   1:  PR[GP1:91,2] = PR[GP1:90,2] + 0.287;
   1:L PR[91] 10mm/sec CNT100;
   1:  PR[GP1:91,1] = PR[GP1:90,1] + -53.304;
   1:  PR[GP1:91,2] = PR[GP1:90,2] + -9.649;
   1:L PR[91] 10mm/sec CNT100;
   1:  PR[GP1:91,1] = PR[GP1:90,1] + -52.837;
   1:  PR[GP1:91,2] = PR[GP1:90,2] + -13.000;
   1:L PR[91] 10mm/sec CNT100;
   1:  PR[GP1:91,1] = PR[GP1:90,1] + -51.484;
   1:  PR[GP1:91,2] = PR[GP1:90,2] + -16.066;
   1:L PR[91] 10mm/sec CNT100;
   1:  PR[GP1:91,1] = PR[GP1:90,1] + -46.658;
   1:  PR[GP1:91,2] = PR[GP1:90,2] + -24.961;
   1:L PR[91] 10mm/sec CNT100;
   1:  PR[GP1:91,1] = PR[GP1:90,1] + -44.364;
   1:  PR[GP1:91,2] = PR[GP1:90,2] + -27.724;
   1:L PR[91] 10mm/sec CNT100;
   1:  PR[GP1:91,1] = PR[GP1:90,1] + -37.102;
   1:  PR[GP1:91,2] = PR[GP1:90,2] + -34.467;
   1:L PR[91] 10mm/sec CNT100;
   1:  PR[GP1:91,1] = PR[GP1:90,1] + -32.633;
   1:  PR[GP1:91,2] = PR[GP1:90,2] + -37.235;
   1:L PR[91] 10mm/sec CNT100;
   1:  PR[GP1:91,1] = PR[GP1:90,1] + -23.806;
   1:  PR[GP1:91,2] = PR[GP1:90,2] + -41.267;
   1:L PR[91] 10mm/sec CNT100;
   1:  PR[GP1:91,1] = PR[GP1:90,1] + -18.131;
   1:  PR[GP1:91,2] = PR[GP1:90,2] + -42.329;
   1:L PR[91] 10mm/sec CNT100;
   1:  PR[GP1:91,1] = PR[GP1:90,1] + -8.768;
   1:  PR[GP1:91,2] = PR[GP1:90,2] + -43.356;
   1:L PR[91] 10mm/sec CNT100;
   1:  PR[GP1:91,1] = PR[GP1:90,1] + -2.914;
   1:  PR[GP1:91,2] = PR[GP1:90,2] + -42.375;
   1:L PR[91] 10mm/sec CNT100;
   1:  PR[GP1:91,1] = PR[GP1:90,1] + -0.261;
   1:  PR[GP1:91,2] = PR[GP1:90,2] + -41.804;
   1:L PR[91] 10mm/sec CNT100;
   1:  PR[GP1:91,1] = PR[GP1:90,1] + 1.954;
   1:  PR[GP1:91,2] = PR[GP1:90,2] + -42.461;
   1:  PR[GP1:91,3] = PR[GP1:90,3] + 101.565;
   1:L PR[91] 10mm/sec CNT100;
   1:  PR[GP1:91,1] = PR[GP1:90,1] + 8.050;
   1:  PR[GP1:91,2] = PR[GP1:90,2] + -43.485;
   1:L PR[91] 10mm/sec CNT100;
   1:  PR[GP1:91,1] = PR[GP1:90,1] + 17.201;
   1:  PR[GP1:91,2] = PR[GP1:90,2] + -42.479;
   1:L PR[91] 10mm/sec CNT100;
   1:  PR[GP1:91,1] = PR[GP1:90,1] + 23.153;
   1:  PR[GP1:91,2] = PR[GP1:90,2] + -41.367;
   1:L PR[91] 10mm/sec CNT100;
   1:  PR[GP1:91,1] = PR[GP1:90,1] + 31.780;
   1:  PR[GP1:91,2] = PR[GP1:90,2] + -37.429;
   1:L PR[91] 10mm/sec CNT100;
   1:  PR[GP1:91,1] = PR[GP1:90,1] + 36.498;
   1:  PR[GP1:91,2] = PR[GP1:90,2] + -34.507;
   1:L PR[91] 10mm/sec CNT100;
   1:  PR[GP1:91,1] = PR[GP1:90,1] + 43.596;
   1:  PR[GP1:91,2] = PR[GP1:90,2] + -27.908;
   1:L PR[91] 10mm/sec CNT100;
   1:  PR[GP1:91,1] = PR[GP1:90,1] + 46.034;
   1:  PR[GP1:91,2] = PR[GP1:90,2] + -24.972;
   1:L PR[91] 10mm/sec CNT100;
   1:  PR[GP1:91,1] = PR[GP1:90,1] + 50.751;
   1:  PR[GP1:91,2] = PR[GP1:90,2] + -16.292;
   1:L PR[91] 10mm/sec CNT100;
   1:  PR[GP1:91,1] = PR[GP1:90,1] + 52.201;
   1:  PR[GP1:91,2] = PR[GP1:90,2] + -13.008;
   1:L PR[91] 10mm/sec CNT100;
   1:  PR[GP1:91,1] = PR[GP1:90,1] + 53.844;
   1:  PR[GP1:91,2] = PR[GP1:90,2] + -3.236;
   1:L PR[91] 10mm/sec CNT100;
   1:  PR[GP1:91,1] = PR[GP1:90,1] + 53.846;
   1:  PR[GP1:91,2] = PR[GP1:90,2] + -2.997;
   1:L PR[91] 10mm/sec CNT100;
   1:  PR[GP1:91,1] = PR[GP1:90,1] + 54.302;
   1:  PR[GP1:91,2] = PR[GP1:90,2] + 0.271;
   1:L PR[91] 10mm/sec CNT100;
   1:  PR[GP1:91,1] = PR[GP1:90,1] + 52.690;
   1:  PR[GP1:91,2] = PR[GP1:90,2] + 10.014;
   1:L PR[91] 10mm/sec CNT100;
   1:  PR[GP1:91,1] = PR[GP1:90,1] + 52.191;
   1:  PR[GP1:91,2] = PR[GP1:90,2] + 13.594;
   1:L PR[91] 10mm/sec CNT100;
   1:  PR[GP1:91,1] = PR[GP1:90,1] + 50.744;
   1:  PR[GP1:91,2] = PR[GP1:90,2] + 16.870;
   1:L PR[91] 10mm/sec CNT100;
   1:  PR[GP1:91,1] = PR[GP1:90,1] + 46.008;
   1:  PR[GP1:91,2] = PR[GP1:90,2] + 25.563;
   1:L PR[91] 10mm/sec CNT100;
   1:  PR[GP1:91,1] = PR[GP1:90,1] + 43.570;
   1:  PR[GP1:91,2] = PR[GP1:90,2] + 28.500;
   1:L PR[91] 10mm/sec CNT100;
   1:  PR[GP1:91,1] = PR[GP1:90,1] + 36.447;
   1:  PR[GP1:91,2] = PR[GP1:90,2] + 35.099;
   1:L PR[91] 10mm/sec CNT100;
   1:  PR[GP1:91,1] = PR[GP1:90,1] + 31.727;
   1:  PR[GP1:91,2] = PR[GP1:90,2] + 38.022;
   1:L PR[91] 10mm/sec CNT100;
   1:  PR[GP1:91,1] = PR[GP1:90,1] + 23.077;
   1:  PR[GP1:91,2] = PR[GP1:90,2] + 41.946;
   1:L PR[91] 10mm/sec CNT100;
   1:  PR[GP1:91,1] = PR[GP1:90,1] + 17.121;
   1:  PR[GP1:91,2] = PR[GP1:90,2] + 43.059;
   1:L PR[91] 10mm/sec CNT100;
   1:  PR[GP1:91,1] = PR[GP1:90,1] + 7.957;
   1:  PR[GP1:91,2] = PR[GP1:90,2] + 44.038;
   1:L PR[91] 10mm/sec CNT100;
   1:  PR[GP1:91,1] = PR[GP1:90,1] + -0.260;
   1:  PR[GP1:91,2] = PR[GP1:90,2] + 42.592;
   1:L PR[91] 10mm/sec CNT100;
   1:  PR[GP1:91,1] = PR[GP1:90,1] + -8.486;
   1:  PR[GP1:91,2] = PR[GP1:90,2] + 44.037;
   1:L PR[91] 10mm/sec CNT100;
   1:  PR[GP1:91,1] = PR[GP1:90,1] + -17.650;
   1:  PR[GP1:91,2] = PR[GP1:90,2] + 43.060;
   1:L PR[91] 10mm/sec CNT100;
   1:  PR[GP1:91,1] = PR[GP1:90,1] + -23.604;
   1:  PR[GP1:91,2] = PR[GP1:90,2] + 41.946;
   1:L PR[91] 10mm/sec CNT100;
   1:  PR[GP1:91,1] = PR[GP1:90,1] + -32.254;
   1:  PR[GP1:91,2] = PR[GP1:90,2] + 38.019;
   1:L PR[91] 10mm/sec CNT100;
   1:  PR[GP1:91,1] = PR[GP1:90,1] + -36.973;
   1:  PR[GP1:91,2] = PR[GP1:90,2] + 35.097;
   1:L PR[91] 10mm/sec CNT100;
   1:  PR[GP1:91,1] = PR[GP1:90,1] + -44.096;
   1:  PR[GP1:91,2] = PR[GP1:90,2] + 28.506;
   1:L PR[91] 10mm/sec CNT100;
   1:  PR[GP1:91,1] = PR[GP1:90,1] + -46.534;
   1:  PR[GP1:91,2] = PR[GP1:90,2] + 25.569;
   1:L PR[91] 10mm/sec CNT100;
   1:  PR[GP1:91,1] = PR[GP1:90,1] + -51.270;
   1:  PR[GP1:91,2] = PR[GP1:90,2] + 16.861;
   1:L PR[91] 10mm/sec CNT100;
   1:  PR[GP1:91,1] = PR[GP1:90,1] + -52.721;
   1:  PR[GP1:91,2] = PR[GP1:90,2] + 13.576;
   1:L PR[91] 10mm/sec CNT100;
   1:  PR[GP1:91,1] = PR[GP1:90,1] + -54.370;
   1:  PR[GP1:91,2] = PR[GP1:90,2] + 3.794;
   1:L PR[91] 10mm/sec CNT100;
   1:  PR[GP1:91,1] = PR[GP1:90,1] + -54.373;
   1:  PR[GP1:91,2] = PR[GP1:90,2] + 3.555;
   1:L PR[91] 10mm/sec CNT100;
   1:  PR[GP1:91,1] = PR[GP1:90,1] + -54.828;
   1:  PR[GP1:91,2] = PR[GP1:90,2] + 0.287;
   1:L PR[91] 10mm/sec CNT100;
   1:  PR[GP1:91,1] = PR[GP1:90,1] + -53.223;
   1:  PR[GP1:91,2] = PR[GP1:90,2] + -9.426;
   1:L PR[91] 10mm/sec CNT100;
   1:  PR[GP1:91,1] = PR[GP1:90,1] + -52.724;
   1:  PR[GP1:91,2] = PR[GP1:90,2] + -13.005;
   1:L PR[91] 10mm/sec CNT100;
   1:  PR[GP1:91,1] = PR[GP1:90,1] + -51.277;
   1:  PR[GP1:91,2] = PR[GP1:90,2] + -16.282;
   1:L PR[91] 10mm/sec CNT100;
   1:  PR[GP1:91,1] = PR[GP1:90,1] + -46.560;
   1:  PR[GP1:91,2] = PR[GP1:90,2] + -24.978;
   1:L PR[91] 10mm/sec CNT100;
   1:  PR[GP1:91,1] = PR[GP1:90,1] + -44.122;
   1:  PR[GP1:91,2] = PR[GP1:90,2] + -27.914;
   1:L PR[91] 10mm/sec CNT100;
   1:  PR[GP1:91,1] = PR[GP1:90,1] + -37.024;
   1:  PR[GP1:91,2] = PR[GP1:90,2] + -34.505;
   1:L PR[91] 10mm/sec CNT100;
   1:  PR[GP1:91,1] = PR[GP1:90,1] + -32.308;
   1:  PR[GP1:91,2] = PR[GP1:90,2] + -37.426;
   1:L PR[91] 10mm/sec CNT100;
   1:  PR[GP1:91,1] = PR[GP1:90,1] + -23.680;
   1:  PR[GP1:91,2] = PR[GP1:90,2] + -41.367;
   1:L PR[91] 10mm/sec CNT100;
   1:  PR[GP1:91,1] = PR[GP1:90,1] + -17.730;
   1:  PR[GP1:91,2] = PR[GP1:90,2] + -42.480;
   1:L PR[91] 10mm/sec CNT100;
   1:  PR[GP1:91,1] = PR[GP1:90,1] + -8.579;
   1:  PR[GP1:91,2] = PR[GP1:90,2] + -43.484;
   1:L PR[91] 10mm/sec CNT100;
   1:  PR[GP1:91,1] = PR[GP1:90,1] + -2.476;
   1:  PR[GP1:91,2] = PR[GP1:90,2] + -42.461;
   1:L PR[91] 10mm/sec CNT100;
   1:  PR[GP1:91,1] = PR[GP1:90,1] + -0.261;
   1:  PR[GP1:91,2] = PR[GP1:90,2] + -41.985;
   1:L PR[91] 10mm/sec CNT100;
   1:  PR[GP1:91,1] = PR[GP1:90,1] + 1.516;
   1:  PR[GP1:91,2] = PR[GP1:90,2] + -42.548;
   1:  PR[GP1:91,3] = PR[GP1:90,3] + 102.175;
   1:L PR[91] 10mm/sec CNT100;
   1:  PR[GP1:91,1] = PR[GP1:90,1] + 7.860;
   1:  PR[GP1:91,2] = PR[GP1:90,2] + -43.613;
   1:L PR[91] 10mm/sec CNT100;
   1:  PR[GP1:91,1] = PR[GP1:90,1] + 16.800;
   1:  PR[GP1:91,2] = PR[GP1:90,2] + -42.631;
   1:L PR[91] 10mm/sec CNT100;
   1:  PR[GP1:91,1] = PR[GP1:90,1] + 23.027;
   1:  PR[GP1:91,2] = PR[GP1:90,2] + -41.467;
   1:L PR[91] 10mm/sec CNT100;
   1:  PR[GP1:91,1] = PR[GP1:90,1] + 31.455;
   1:  PR[GP1:91,2] = PR[GP1:90,2] + -37.620;
   1:L PR[91] 10mm/sec CNT100;
   1:  PR[GP1:91,1] = PR[GP1:90,1] + 36.419;
   1:  PR[GP1:91,2] = PR[GP1:90,2] + -34.545;
   1:L PR[91] 10mm/sec CNT100;
   1:  PR[GP1:91,1] = PR[GP1:90,1] + 43.355;
   1:  PR[GP1:91,2] = PR[GP1:90,2] + -28.098;
   1:L PR[91] 10mm/sec CNT100;
   1:  PR[GP1:91,1] = PR[GP1:90,1] + 45.936;
   1:  PR[GP1:91,2] = PR[GP1:90,2] + -24.988;
   1:L PR[91] 10mm/sec CNT100;
   1:  PR[GP1:91,1] = PR[GP1:90,1] + 50.545;
   1:  PR[GP1:91,2] = PR[GP1:90,2] + -16.509;
   1:L PR[91] 10mm/sec CNT100;
   1:  PR[GP1:91,1] = PR[GP1:90,1] + 52.088;
   1:  PR[GP1:91,2] = PR[GP1:90,2] + -13.013;
   1:L PR[91] 10mm/sec CNT100;
   1:  PR[GP1:91,1] = PR[GP1:90,1] + 53.693;
   1:  PR[GP1:91,2] = PR[GP1:90,2] + -3.467;
   1:L PR[91] 10mm/sec CNT100;
   1:  PR[GP1:91,1] = PR[GP1:90,1] + 53.695;
   1:  PR[GP1:91,2] = PR[GP1:90,2] + -3.233;
   1:L PR[91] 10mm/sec CNT100;
   1:  PR[GP1:91,1] = PR[GP1:90,1] + 54.184;
   1:  PR[GP1:91,2] = PR[GP1:90,2] + 0.271;
   1:L PR[91] 10mm/sec CNT100;
   1:  PR[GP1:91,1] = PR[GP1:90,1] + 52.609;
   1:  PR[GP1:91,2] = PR[GP1:90,2] + 9.790;
   1:L PR[91] 10mm/sec CNT100;
   1:  PR[GP1:91,1] = PR[GP1:90,1] + 52.078;
   1:  PR[GP1:91,2] = PR[GP1:90,2] + 13.598;
   1:L PR[91] 10mm/sec CNT100;
   1:  PR[GP1:91,1] = PR[GP1:90,1] + 50.538;
   1:  PR[GP1:91,2] = PR[GP1:90,2] + 17.086;
   1:L PR[91] 10mm/sec CNT100;
   1:  PR[GP1:91,1] = PR[GP1:90,1] + 45.911;
   1:  PR[GP1:91,2] = PR[GP1:90,2] + 25.579;
   1:L PR[91] 10mm/sec CNT100;
   1:  PR[GP1:91,1] = PR[GP1:90,1] + 43.329;
   1:  PR[GP1:91,2] = PR[GP1:90,2] + 28.690;
   1:L PR[91] 10mm/sec CNT100;
   1:  PR[GP1:91,1] = PR[GP1:90,1] + 36.370;
   1:  PR[GP1:91,2] = PR[GP1:90,2] + 35.136;
   1:L PR[91] 10mm/sec CNT100;
   1:  PR[GP1:91,1] = PR[GP1:90,1] + 31.403;
   1:  PR[GP1:91,2] = PR[GP1:90,2] + 38.212;
   1:L PR[91] 10mm/sec CNT100;
   1:  PR[GP1:91,1] = PR[GP1:90,1] + 22.953;
   1:  PR[GP1:91,2] = PR[GP1:90,2] + 42.046;
   1:L PR[91] 10mm/sec CNT100;
   1:  PR[GP1:91,1] = PR[GP1:90,1] + 16.722;
   1:  PR[GP1:91,2] = PR[GP1:90,2] + 43.210;
   1:L PR[91] 10mm/sec CNT100;
   1:  PR[GP1:91,1] = PR[GP1:90,1] + 7.770;
   1:  PR[GP1:91,2] = PR[GP1:90,2] + 44.166;
   1:L PR[91] 10mm/sec CNT100;
   1:  PR[GP1:91,1] = PR[GP1:90,1] + -0.260;
   1:  PR[GP1:91,2] = PR[GP1:90,2] + 42.754;
   1:L PR[91] 10mm/sec CNT100;
   1:  PR[GP1:91,1] = PR[GP1:90,1] + -8.299;
   1:  PR[GP1:91,2] = PR[GP1:90,2] + 44.166;
   1:L PR[91] 10mm/sec CNT100;
   1:  PR[GP1:91,1] = PR[GP1:90,1] + -17.251;
   1:  PR[GP1:91,2] = PR[GP1:90,2] + 43.211;
   1:L PR[91] 10mm/sec CNT100;
   1:  PR[GP1:91,1] = PR[GP1:90,1] + -23.480;
   1:  PR[GP1:91,2] = PR[GP1:90,2] + 42.046;
   1:L PR[91] 10mm/sec CNT100;
   1:  PR[GP1:91,1] = PR[GP1:90,1] + -31.930;
   1:  PR[GP1:91,2] = PR[GP1:90,2] + 38.210;
   1:L PR[91] 10mm/sec CNT100;
   1:  PR[GP1:91,1] = PR[GP1:90,1] + -36.896;
   1:  PR[GP1:91,2] = PR[GP1:90,2] + 35.135;
   1:L PR[91] 10mm/sec CNT100;
   1:  PR[GP1:91,1] = PR[GP1:90,1] + -43.855;
   1:  PR[GP1:91,2] = PR[GP1:90,2] + 28.695;
   1:L PR[91] 10mm/sec CNT100;
   1:  PR[GP1:91,1] = PR[GP1:90,1] + -46.437;
   1:  PR[GP1:91,2] = PR[GP1:90,2] + 25.585;
   1:L PR[91] 10mm/sec CNT100;
   1:  PR[GP1:91,1] = PR[GP1:90,1] + -51.064;
   1:  PR[GP1:91,2] = PR[GP1:90,2] + 17.077;
   1:L PR[91] 10mm/sec CNT100;
   1:  PR[GP1:91,1] = PR[GP1:90,1] + -52.608;
   1:  PR[GP1:91,2] = PR[GP1:90,2] + 13.580;
   1:L PR[91] 10mm/sec CNT100;
   1:  PR[GP1:91,1] = PR[GP1:90,1] + -54.219;
   1:  PR[GP1:91,2] = PR[GP1:90,2] + 4.025;
   1:L PR[91] 10mm/sec CNT100;
   1:  PR[GP1:91,1] = PR[GP1:90,1] + -54.222;
   1:  PR[GP1:91,2] = PR[GP1:90,2] + 3.792;
   1:L PR[91] 10mm/sec CNT100;
   1:  PR[GP1:91,1] = PR[GP1:90,1] + -54.710;
   1:  PR[GP1:91,2] = PR[GP1:90,2] + 0.287;
   1:L PR[91] 10mm/sec CNT100;
   1:  PR[GP1:91,1] = PR[GP1:90,1] + -53.142;
   1:  PR[GP1:91,2] = PR[GP1:90,2] + -9.202;
   1:L PR[91] 10mm/sec CNT100;
   1:  PR[GP1:91,1] = PR[GP1:90,1] + -52.611;
   1:  PR[GP1:91,2] = PR[GP1:90,2] + -13.011;
   1:L PR[91] 10mm/sec CNT100;
   1:  PR[GP1:91,1] = PR[GP1:90,1] + -51.071;
   1:  PR[GP1:91,2] = PR[GP1:90,2] + -16.499;
   1:L PR[91] 10mm/sec CNT100;
   1:  PR[GP1:91,1] = PR[GP1:90,1] + -46.462;
   1:  PR[GP1:91,2] = PR[GP1:90,2] + -24.994;
   1:L PR[91] 10mm/sec CNT100;
   1:  PR[GP1:91,1] = PR[GP1:90,1] + -43.881;
   1:  PR[GP1:91,2] = PR[GP1:90,2] + -28.104;
   1:L PR[91] 10mm/sec CNT100;
   1:  PR[GP1:91,1] = PR[GP1:90,1] + -36.945;
   1:  PR[GP1:91,2] = PR[GP1:90,2] + -34.544;
   1:L PR[91] 10mm/sec CNT100;
   1:  PR[GP1:91,1] = PR[GP1:90,1] + -31.982;
   1:  PR[GP1:91,2] = PR[GP1:90,2] + -37.617;
   1:L PR[91] 10mm/sec CNT100;
   1:  PR[GP1:91,1] = PR[GP1:90,1] + -23.554;
   1:  PR[GP1:91,2] = PR[GP1:90,2] + -41.468;
   1:L PR[91] 10mm/sec CNT100;
   1:  PR[GP1:91,1] = PR[GP1:90,1] + -17.330;
   1:  PR[GP1:91,2] = PR[GP1:90,2] + -42.632;
   1:L PR[91] 10mm/sec CNT100;
   1:  PR[GP1:91,1] = PR[GP1:90,1] + -8.390;
   1:  PR[GP1:91,2] = PR[GP1:90,2] + -43.613;
   1:L PR[91] 10mm/sec CNT100;
   1:  PR[GP1:91,1] = PR[GP1:90,1] + -2.038;
   1:  PR[GP1:91,2] = PR[GP1:90,2] + -42.548;
   1:L PR[91] 10mm/sec CNT100;
   1:  PR[GP1:91,1] = PR[GP1:90,1] + -0.261;
   1:  PR[GP1:91,2] = PR[GP1:90,2] + -42.166;
   1:L PR[91] 10mm/sec CNT100;
   1:  PR[GP1:91,1] = PR[GP1:90,1] + 1.079;
   1:  PR[GP1:91,2] = PR[GP1:90,2] + -42.635;
   1:  PR[GP1:91,3] = PR[GP1:90,3] + 102.785;
   1:L PR[91] 10mm/sec CNT100;
   1:  PR[GP1:91,1] = PR[GP1:90,1] + 7.671;
   1:  PR[GP1:91,2] = PR[GP1:90,2] + -43.742;
   1:L PR[91] 10mm/sec CNT100;
   1:  PR[GP1:91,1] = PR[GP1:90,1] + 16.400;
   1:  PR[GP1:91,2] = PR[GP1:90,2] + -42.783;
   1:L PR[91] 10mm/sec CNT100;
   1:  PR[GP1:91,1] = PR[GP1:90,1] + 22.900;
   1:  PR[GP1:91,2] = PR[GP1:90,2] + -41.568;
   1:L PR[91] 10mm/sec CNT100;
   1:  PR[GP1:91,1] = PR[GP1:90,1] + 31.130;
   1:  PR[GP1:91,2] = PR[GP1:90,2] + -37.811;
   1:L PR[91] 10mm/sec CNT100;
   1:  PR[GP1:91,1] = PR[GP1:90,1] + 36.341;
   1:  PR[GP1:91,2] = PR[GP1:90,2] + -34.584;
   1:L PR[91] 10mm/sec CNT100;
   1:  PR[GP1:91,1] = PR[GP1:90,1] + 43.113;
   1:  PR[GP1:91,2] = PR[GP1:90,2] + -28.289;
   1:L PR[91] 10mm/sec CNT100;
   1:  PR[GP1:91,1] = PR[GP1:90,1] + 45.839;
   1:  PR[GP1:91,2] = PR[GP1:90,2] + -25.005;
   1:L PR[91] 10mm/sec CNT100;
   1:  PR[GP1:91,1] = PR[GP1:90,1] + 50.339;
   1:  PR[GP1:91,2] = PR[GP1:90,2] + -16.725;
   1:L PR[91] 10mm/sec CNT100;
   1:  PR[GP1:91,1] = PR[GP1:90,1] + 51.975;
   1:  PR[GP1:91,2] = PR[GP1:90,2] + -13.018;
   1:L PR[91] 10mm/sec CNT100;
   1:  PR[GP1:91,1] = PR[GP1:90,1] + 53.542;
   1:  PR[GP1:91,2] = PR[GP1:90,2] + -3.698;
   1:L PR[91] 10mm/sec CNT100;
   1:  PR[GP1:91,1] = PR[GP1:90,1] + 53.544;
   1:  PR[GP1:91,2] = PR[GP1:90,2] + -3.470;
   1:L PR[91] 10mm/sec CNT100;
   1:  PR[GP1:91,1] = PR[GP1:90,1] + 54.066;
   1:  PR[GP1:91,2] = PR[GP1:90,2] + 0.271;
   1:L PR[91] 10mm/sec CNT100;
   1:  PR[GP1:91,1] = PR[GP1:90,1] + 52.528;
   1:  PR[GP1:91,2] = PR[GP1:90,2] + 9.566;
   1:L PR[91] 10mm/sec CNT100;
   1:  PR[GP1:91,1] = PR[GP1:90,1] + 51.965;
   1:  PR[GP1:91,2] = PR[GP1:90,2] + 13.603;
   1:L PR[91] 10mm/sec CNT100;
   1:  PR[GP1:91,1] = PR[GP1:90,1] + 50.332;
   1:  PR[GP1:91,2] = PR[GP1:90,2] + 17.302;
   1:L PR[91] 10mm/sec CNT100;
   1:  PR[GP1:91,1] = PR[GP1:90,1] + 45.814;
   1:  PR[GP1:91,2] = PR[GP1:90,2] + 25.595;
   1:L PR[91] 10mm/sec CNT100;
   1:  PR[GP1:91,1] = PR[GP1:90,1] + 43.088;
   1:  PR[GP1:91,2] = PR[GP1:90,2] + 28.879;
   1:L PR[91] 10mm/sec CNT100;
   1:  PR[GP1:91,1] = PR[GP1:90,1] + 36.293;
   1:  PR[GP1:91,2] = PR[GP1:90,2] + 35.174;
   1:L PR[91] 10mm/sec CNT100;
   1:  PR[GP1:91,1] = PR[GP1:90,1] + 31.079;
   1:  PR[GP1:91,2] = PR[GP1:90,2] + 38.403;
   1:L PR[91] 10mm/sec CNT100;
   1:  PR[GP1:91,1] = PR[GP1:90,1] + 22.828;
   1:  PR[GP1:91,2] = PR[GP1:90,2] + 42.146;
   1:L PR[91] 10mm/sec CNT100;
   1:  PR[GP1:91,1] = PR[GP1:90,1] + 16.324;
   1:  PR[GP1:91,2] = PR[GP1:90,2] + 43.361;
   1:L PR[91] 10mm/sec CNT100;
   1:  PR[GP1:91,1] = PR[GP1:90,1] + 7.583;
   1:  PR[GP1:91,2] = PR[GP1:90,2] + 44.295;
   1:L PR[91] 10mm/sec CNT100;
   1:  PR[GP1:91,1] = PR[GP1:90,1] + -0.260;
   1:  PR[GP1:91,2] = PR[GP1:90,2] + 42.915;
   1:L PR[91] 10mm/sec CNT100;
   1:  PR[GP1:91,1] = PR[GP1:90,1] + -8.112;
   1:  PR[GP1:91,2] = PR[GP1:90,2] + 44.294;
   1:L PR[91] 10mm/sec CNT100;
   1:  PR[GP1:91,1] = PR[GP1:90,1] + -16.853;
   1:  PR[GP1:91,2] = PR[GP1:90,2] + 43.362;
   1:L PR[91] 10mm/sec CNT100;
   1:  PR[GP1:91,1] = PR[GP1:90,1] + -23.355;
   1:  PR[GP1:91,2] = PR[GP1:90,2] + 42.146;
   1:L PR[91] 10mm/sec CNT100;
   1:  PR[GP1:91,1] = PR[GP1:90,1] + -31.606;
   1:  PR[GP1:91,2] = PR[GP1:90,2] + 38.400;
   1:L PR[91] 10mm/sec CNT100;
   1:  PR[GP1:91,1] = PR[GP1:90,1] + -36.818;
   1:  PR[GP1:91,2] = PR[GP1:90,2] + 35.172;
   1:L PR[91] 10mm/sec CNT100;
   1:  PR[GP1:91,1] = PR[GP1:90,1] + -43.613;
   1:  PR[GP1:91,2] = PR[GP1:90,2] + 28.885;
   1:L PR[91] 10mm/sec CNT100;
   1:  PR[GP1:91,1] = PR[GP1:90,1] + -46.340;
   1:  PR[GP1:91,2] = PR[GP1:90,2] + 25.601;
   1:L PR[91] 10mm/sec CNT100;
   1:  PR[GP1:91,1] = PR[GP1:90,1] + -50.858;
   1:  PR[GP1:91,2] = PR[GP1:90,2] + 17.293;
   1:L PR[91] 10mm/sec CNT100;
   1:  PR[GP1:91,1] = PR[GP1:90,1] + -52.495;
   1:  PR[GP1:91,2] = PR[GP1:90,2] + 13.585;
   1:L PR[91] 10mm/sec CNT100;
   1:  PR[GP1:91,1] = PR[GP1:90,1] + -54.068;
   1:  PR[GP1:91,2] = PR[GP1:90,2] + 4.256;
   1:L PR[91] 10mm/sec CNT100;
   1:  PR[GP1:91,1] = PR[GP1:90,1] + -54.071;
   1:  PR[GP1:91,2] = PR[GP1:90,2] + 4.028;
   1:L PR[91] 10mm/sec CNT100;
   1:  PR[GP1:91,1] = PR[GP1:90,1] + -54.592;
   1:  PR[GP1:91,2] = PR[GP1:90,2] + 0.287;
   1:L PR[91] 10mm/sec CNT100;
   1:  PR[GP1:91,1] = PR[GP1:90,1] + -53.061;
   1:  PR[GP1:91,2] = PR[GP1:90,2] + -8.979;
   1:L PR[91] 10mm/sec CNT100;
   1:  PR[GP1:91,1] = PR[GP1:90,1] + -52.498;
   1:  PR[GP1:91,2] = PR[GP1:90,2] + -13.016;
   1:L PR[91] 10mm/sec CNT100;
   1:  PR[GP1:91,1] = PR[GP1:90,1] + -50.865;
   1:  PR[GP1:91,2] = PR[GP1:90,2] + -16.715;
   1:L PR[91] 10mm/sec CNT100;
   1:  PR[GP1:91,1] = PR[GP1:90,1] + -46.365;
   1:  PR[GP1:91,2] = PR[GP1:90,2] + -25.011;
   1:L PR[91] 10mm/sec CNT100;
   1:  PR[GP1:91,1] = PR[GP1:90,1] + -43.639;
   1:  PR[GP1:91,2] = PR[GP1:90,2] + -28.294;
   1:L PR[91] 10mm/sec CNT100;
   1:  PR[GP1:91,1] = PR[GP1:90,1] + -36.867;
   1:  PR[GP1:91,2] = PR[GP1:90,2] + -34.582;
   1:L PR[91] 10mm/sec CNT100;
   1:  PR[GP1:91,1] = PR[GP1:90,1] + -31.657;
   1:  PR[GP1:91,2] = PR[GP1:90,2] + -37.809;
   1:L PR[91] 10mm/sec CNT100;
   1:  PR[GP1:91,1] = PR[GP1:90,1] + -23.428;
   1:  PR[GP1:91,2] = PR[GP1:90,2] + -41.568;
   1:L PR[91] 10mm/sec CNT100;
   1:  PR[GP1:91,1] = PR[GP1:90,1] + -16.930;
   1:  PR[GP1:91,2] = PR[GP1:90,2] + -42.783;
   1:L PR[91] 10mm/sec CNT100;
   1:  PR[GP1:91,1] = PR[GP1:90,1] + -8.201;
   1:  PR[GP1:91,2] = PR[GP1:90,2] + -43.741;
   1:L PR[91] 10mm/sec CNT100;
   1:  PR[GP1:91,1] = PR[GP1:90,1] + -1.600;
   1:  PR[GP1:91,2] = PR[GP1:90,2] + -42.635;
   1:L PR[91] 10mm/sec CNT100;
   1:  PR[GP1:91,1] = PR[GP1:90,1] + -0.261;
   1:  PR[GP1:91,2] = PR[GP1:90,2] + -42.347;
   1:L PR[91] 10mm/sec CNT100;
   1:  PR[GP1:91,1] = PR[GP1:90,1] + 0.641;
   1:  PR[GP1:91,2] = PR[GP1:90,2] + -42.722;
   1:  PR[GP1:91,3] = PR[GP1:90,3] + 103.395;
   1:L PR[91] 10mm/sec CNT100;
   1:  PR[GP1:91,1] = PR[GP1:90,1] + 7.482;
   1:  PR[GP1:91,2] = PR[GP1:90,2] + -43.870;
   1:L PR[91] 10mm/sec CNT100;
   1:  PR[GP1:91,1] = PR[GP1:90,1] + 15.999;
   1:  PR[GP1:91,2] = PR[GP1:90,2] + -42.934;
   1:L PR[91] 10mm/sec CNT100;
   1:  PR[GP1:91,1] = PR[GP1:90,1] + 22.774;
   1:  PR[GP1:91,2] = PR[GP1:90,2] + -41.668;
   1:L PR[91] 10mm/sec CNT100;
   1:  PR[GP1:91,1] = PR[GP1:90,1] + 30.804;
   1:  PR[GP1:91,2] = PR[GP1:90,2] + -38.002;
   1:L PR[91] 10mm/sec CNT100;
   1:  PR[GP1:91,1] = PR[GP1:90,1] + 36.263;
   1:  PR[GP1:91,2] = PR[GP1:90,2] + -34.622;
   1:L PR[91] 10mm/sec CNT100;
   1:  PR[GP1:91,1] = PR[GP1:90,1] + 42.871;
   1:  PR[GP1:91,2] = PR[GP1:90,2] + -28.479;
   1:L PR[91] 10mm/sec CNT100;
   1:  PR[GP1:91,1] = PR[GP1:90,1] + 45.741;
   1:  PR[GP1:91,2] = PR[GP1:90,2] + -25.022;
   1:L PR[91] 10mm/sec CNT100;
   1:  PR[GP1:91,1] = PR[GP1:90,1] + 50.133;
   1:  PR[GP1:91,2] = PR[GP1:90,2] + -16.941;
   1:L PR[91] 10mm/sec CNT100;
   1:  PR[GP1:91,1] = PR[GP1:90,1] + 51.862;
   1:  PR[GP1:91,2] = PR[GP1:90,2] + -13.023;
   1:L PR[91] 10mm/sec CNT100;
   1:  PR[GP1:91,1] = PR[GP1:90,1] + 53.391;
   1:  PR[GP1:91,2] = PR[GP1:90,2] + -3.928;
   1:L PR[91] 10mm/sec CNT100;
   1:  PR[GP1:91,1] = PR[GP1:90,1] + 53.393;
   1:  PR[GP1:91,2] = PR[GP1:90,2] + -3.706;
   1:L PR[91] 10mm/sec CNT100;
   1:  PR[GP1:91,1] = PR[GP1:90,1] + 53.948;
   1:  PR[GP1:91,2] = PR[GP1:90,2] + 0.271;
   1:L PR[91] 10mm/sec CNT100;
   1:  PR[GP1:91,1] = PR[GP1:90,1] + 52.447;
   1:  PR[GP1:91,2] = PR[GP1:90,2] + 9.341;
   1:L PR[91] 10mm/sec CNT100;
   1:  PR[GP1:91,1] = PR[GP1:90,1] + 51.852;
   1:  PR[GP1:91,2] = PR[GP1:90,2] + 13.608;
   1:L PR[91] 10mm/sec CNT100;
   1:  PR[GP1:91,1] = PR[GP1:90,1] + 50.126;
   1:  PR[GP1:91,2] = PR[GP1:90,2] + 17.518;
   1:L PR[91] 10mm/sec CNT100;
   1:  PR[GP1:91,1] = PR[GP1:90,1] + 45.717;
   1:  PR[GP1:91,2] = PR[GP1:90,2] + 25.611;
   1:L PR[91] 10mm/sec CNT100;
   1:  PR[GP1:91,1] = PR[GP1:90,1] + 42.846;
   1:  PR[GP1:91,2] = PR[GP1:90,2] + 29.069;
   1:L PR[91] 10mm/sec CNT100;
   1:  PR[GP1:91,1] = PR[GP1:90,1] + 36.215;
   1:  PR[GP1:91,2] = PR[GP1:90,2] + 35.211;
   1:L PR[91] 10mm/sec CNT100;
   1:  PR[GP1:91,1] = PR[GP1:90,1] + 30.755;
   1:  PR[GP1:91,2] = PR[GP1:90,2] + 38.593;
   1:L PR[91] 10mm/sec CNT100;
   1:  PR[GP1:91,1] = PR[GP1:90,1] + 22.704;
   1:  PR[GP1:91,2] = PR[GP1:90,2] + 42.245;
   1:L PR[91] 10mm/sec CNT100;
   1:  PR[GP1:91,1] = PR[GP1:90,1] + 15.925;
   1:  PR[GP1:91,2] = PR[GP1:90,2] + 43.512;
   1:L PR[91] 10mm/sec CNT100;
   1:  PR[GP1:91,1] = PR[GP1:90,1] + 7.396;
   1:  PR[GP1:91,2] = PR[GP1:90,2] + 44.423;
   1:L PR[91] 10mm/sec CNT100;
   1:  PR[GP1:91,1] = PR[GP1:90,1] + -0.260;
   1:  PR[GP1:91,2] = PR[GP1:90,2] + 43.077;
   1:L PR[91] 10mm/sec CNT100;
   1:  PR[GP1:91,1] = PR[GP1:90,1] + -7.925;
   1:  PR[GP1:91,2] = PR[GP1:90,2] + 44.423;
   1:L PR[91] 10mm/sec CNT100;
   1:  PR[GP1:91,1] = PR[GP1:90,1] + -16.454;
   1:  PR[GP1:91,2] = PR[GP1:90,2] + 43.513;
   1:L PR[91] 10mm/sec CNT100;
   1:  PR[GP1:91,1] = PR[GP1:90,1] + -23.231;
   1:  PR[GP1:91,2] = PR[GP1:90,2] + 42.246;
   1:L PR[91] 10mm/sec CNT100;
   1:  PR[GP1:91,1] = PR[GP1:90,1] + -31.282;
   1:  PR[GP1:91,2] = PR[GP1:90,2] + 38.591;
   1:L PR[91] 10mm/sec CNT100;
   1:  PR[GP1:91,1] = PR[GP1:90,1] + -36.741;
   1:  PR[GP1:91,2] = PR[GP1:90,2] + 35.210;
   1:L PR[91] 10mm/sec CNT100;
   1:  PR[GP1:91,1] = PR[GP1:90,1] + -43.372;
   1:  PR[GP1:91,2] = PR[GP1:90,2] + 29.074;
   1:L PR[91] 10mm/sec CNT100;
   1:  PR[GP1:91,1] = PR[GP1:90,1] + -46.243;
   1:  PR[GP1:91,2] = PR[GP1:90,2] + 25.616;
   1:L PR[91] 10mm/sec CNT100;
   1:  PR[GP1:91,1] = PR[GP1:90,1] + -50.652;
   1:  PR[GP1:91,2] = PR[GP1:90,2] + 17.509;
   1:L PR[91] 10mm/sec CNT100;
   1:  PR[GP1:91,1] = PR[GP1:90,1] + -52.382;
   1:  PR[GP1:91,2] = PR[GP1:90,2] + 13.590;
   1:L PR[91] 10mm/sec CNT100;
   1:  PR[GP1:91,1] = PR[GP1:90,1] + -53.917;
   1:  PR[GP1:91,2] = PR[GP1:90,2] + 4.486;
   1:L PR[91] 10mm/sec CNT100;
   1:  PR[GP1:91,1] = PR[GP1:90,1] + -53.920;
   1:  PR[GP1:91,2] = PR[GP1:90,2] + 4.264;
   1:L PR[91] 10mm/sec CNT100;
   1:  PR[GP1:91,1] = PR[GP1:90,1] + -54.474;
   1:  PR[GP1:91,2] = PR[GP1:90,2] + 0.287;
   1:L PR[91] 10mm/sec CNT100;
   1:  PR[GP1:91,1] = PR[GP1:90,1] + -52.980;
   1:  PR[GP1:91,2] = PR[GP1:90,2] + -8.755;
   1:L PR[91] 10mm/sec CNT100;
   1:  PR[GP1:91,1] = PR[GP1:90,1] + -52.385;
   1:  PR[GP1:91,2] = PR[GP1:90,2] + -13.021;
   1:L PR[91] 10mm/sec CNT100;
   1:  PR[GP1:91,1] = PR[GP1:90,1] + -50.659;
   1:  PR[GP1:91,2] = PR[GP1:90,2] + -16.932;
   1:L PR[91] 10mm/sec CNT100;
   1:  PR[GP1:91,1] = PR[GP1:90,1] + -46.267;
   1:  PR[GP1:91,2] = PR[GP1:90,2] + -25.027;
   1:L PR[91] 10mm/sec CNT100;
   1:  PR[GP1:91,1] = PR[GP1:90,1] + -43.397;
   1:  PR[GP1:91,2] = PR[GP1:90,2] + -28.485;
   1:L PR[91] 10mm/sec CNT100;
   1:  PR[GP1:91,1] = PR[GP1:90,1] + -36.789;
   1:  PR[GP1:91,2] = PR[GP1:90,2] + -34.620;
   1:L PR[91] 10mm/sec CNT100;
   1:  PR[GP1:91,1] = PR[GP1:90,1] + -31.332;
   1:  PR[GP1:91,2] = PR[GP1:90,2] + -38.000;
   1:L PR[91] 10mm/sec CNT100;
   1:  PR[GP1:91,1] = PR[GP1:90,1] + -23.302;
   1:  PR[GP1:91,2] = PR[GP1:90,2] + -41.668;
   1:L PR[91] 10mm/sec CNT100;
   1:  PR[GP1:91,1] = PR[GP1:90,1] + -16.529;
   1:  PR[GP1:91,2] = PR[GP1:90,2] + -42.935;
   1:L PR[91] 10mm/sec CNT100;
   1:  PR[GP1:91,1] = PR[GP1:90,1] + -8.011;
   1:  PR[GP1:91,2] = PR[GP1:90,2] + -43.870;
   1:L PR[91] 10mm/sec CNT100;
   1:  PR[GP1:91,1] = PR[GP1:90,1] + -1.162;
   1:  PR[GP1:91,2] = PR[GP1:90,2] + -42.722;
   1:L PR[91] 10mm/sec CNT100;
   1:  PR[GP1:91,1] = PR[GP1:90,1] + -0.261;
   1:  PR[GP1:91,2] = PR[GP1:90,2] + -42.528;
   1:L PR[91] 10mm/sec CNT100;
   1:  PR[GP1:91,1] = PR[GP1:90,1] + 0.203;
   1:  PR[GP1:91,2] = PR[GP1:90,2] + -42.808;
   1:  PR[GP1:91,3] = PR[GP1:90,3] + 104.005;
   1:L PR[91] 10mm/sec CNT100;
   1:  PR[GP1:91,1] = PR[GP1:90,1] + 7.292;
   1:  PR[GP1:91,2] = PR[GP1:90,2] + -43.999;
   1:L PR[91] 10mm/sec CNT100;
   1:  PR[GP1:91,1] = PR[GP1:90,1] + 15.599;
   1:  PR[GP1:91,2] = PR[GP1:90,2] + -43.086;
   1:L PR[91] 10mm/sec CNT100;
   1:  PR[GP1:91,1] = PR[GP1:90,1] + 22.648;
   1:  PR[GP1:91,2] = PR[GP1:90,2] + -41.768;
   1:L PR[91] 10mm/sec CNT100;
   1:  PR[GP1:91,1] = PR[GP1:90,1] + 30.479;
   1:  PR[GP1:91,2] = PR[GP1:90,2] + -38.194;
   1:L PR[91] 10mm/sec CNT100;
   1:  PR[GP1:91,1] = PR[GP1:90,1] + 36.184;
   1:  PR[GP1:91,2] = PR[GP1:90,2] + -34.660;
   1:L PR[91] 10mm/sec CNT100;
   1:  PR[GP1:91,1] = PR[GP1:90,1] + 42.629;
   1:  PR[GP1:91,2] = PR[GP1:90,2] + -28.669;
   1:L PR[91] 10mm/sec CNT100;
   1:  PR[GP1:91,1] = PR[GP1:90,1] + 45.643;
   1:  PR[GP1:91,2] = PR[GP1:90,2] + -25.038;
   1:L PR[91] 10mm/sec CNT100;
   1:  PR[GP1:91,1] = PR[GP1:90,1] + 49.926;
   1:  PR[GP1:91,2] = PR[GP1:90,2] + -17.157;
   1:L PR[91] 10mm/sec CNT100;
   1:  PR[GP1:91,1] = PR[GP1:90,1] + 51.749;
   1:  PR[GP1:91,2] = PR[GP1:90,2] + -13.028;
   1:L PR[91] 10mm/sec CNT100;
   1:  PR[GP1:91,1] = PR[GP1:90,1] + 53.240;
   1:  PR[GP1:91,2] = PR[GP1:90,2] + -4.159;
   1:L PR[91] 10mm/sec CNT100;
   1:  PR[GP1:91,1] = PR[GP1:90,1] + 53.242;
   1:  PR[GP1:91,2] = PR[GP1:90,2] + -3.942;
   1:L PR[91] 10mm/sec CNT100;
   1:  PR[GP1:91,1] = PR[GP1:90,1] + 53.830;
   1:  PR[GP1:91,2] = PR[GP1:90,2] + 0.271;
   1:L PR[91] 10mm/sec CNT100;
   1:  PR[GP1:91,1] = PR[GP1:90,1] + 52.366;
   1:  PR[GP1:91,2] = PR[GP1:90,2] + 9.117;
   1:L PR[91] 10mm/sec CNT100;
   1:  PR[GP1:91,1] = PR[GP1:90,1] + 51.740;
   1:  PR[GP1:91,2] = PR[GP1:90,2] + 13.612;
   1:L PR[91] 10mm/sec CNT100;
   1:  PR[GP1:91,1] = PR[GP1:90,1] + 49.920;
   1:  PR[GP1:91,2] = PR[GP1:90,2] + 17.734;
   1:L PR[91] 10mm/sec CNT100;
   1:  PR[GP1:91,1] = PR[GP1:90,1] + 45.620;
   1:  PR[GP1:91,2] = PR[GP1:90,2] + 25.626;
   1:L PR[91] 10mm/sec CNT100;
   1:  PR[GP1:91,1] = PR[GP1:90,1] + 42.605;
   1:  PR[GP1:91,2] = PR[GP1:90,2] + 29.258;
   1:L PR[91] 10mm/sec CNT100;
   1:  PR[GP1:91,1] = PR[GP1:90,1] + 36.138;
   1:  PR[GP1:91,2] = PR[GP1:90,2] + 35.249;
   1:L PR[91] 10mm/sec CNT100;
   1:  PR[GP1:91,1] = PR[GP1:90,1] + 30.431;
   1:  PR[GP1:91,2] = PR[GP1:90,2] + 38.783;
   1:L PR[91] 10mm/sec CNT100;
   1:  PR[GP1:91,1] = PR[GP1:90,1] + 22.579;
   1:  PR[GP1:91,2] = PR[GP1:90,2] + 42.345;
   1:L PR[91] 10mm/sec CNT100;
   1:  PR[GP1:91,1] = PR[GP1:90,1] + 15.526;
   1:  PR[GP1:91,2] = PR[GP1:90,2] + 43.664;
   1:L PR[91] 10mm/sec CNT100;
   1:  PR[GP1:91,1] = PR[GP1:90,1] + 7.209;
   1:  PR[GP1:91,2] = PR[GP1:90,2] + 44.552;
   1:L PR[91] 10mm/sec CNT100;
   1:  PR[GP1:91,1] = PR[GP1:90,1] + -0.260;
   1:  PR[GP1:91,2] = PR[GP1:90,2] + 43.238;
   1:L PR[91] 10mm/sec CNT100;
   1:  PR[GP1:91,1] = PR[GP1:90,1] + -7.738;
   1:  PR[GP1:91,2] = PR[GP1:90,2] + 44.552;
   1:L PR[91] 10mm/sec CNT100;
   1:  PR[GP1:91,1] = PR[GP1:90,1] + -16.056;
   1:  PR[GP1:91,2] = PR[GP1:90,2] + 43.664;
   1:L PR[91] 10mm/sec CNT100;
   1:  PR[GP1:91,1] = PR[GP1:90,1] + -23.106;
   1:  PR[GP1:91,2] = PR[GP1:90,2] + 42.346;
   1:L PR[91] 10mm/sec CNT100;
   1:  PR[GP1:91,1] = PR[GP1:90,1] + -30.958;
   1:  PR[GP1:91,2] = PR[GP1:90,2] + 38.781;
   1:L PR[91] 10mm/sec CNT100;
   1:  PR[GP1:91,1] = PR[GP1:90,1] + -36.664;
   1:  PR[GP1:91,2] = PR[GP1:90,2] + 35.247;
   1:L PR[91] 10mm/sec CNT100;
   1:  PR[GP1:91,1] = PR[GP1:90,1] + -43.131;
   1:  PR[GP1:91,2] = PR[GP1:90,2] + 29.264;
   1:L PR[91] 10mm/sec CNT100;
   1:  PR[GP1:91,1] = PR[GP1:90,1] + -46.146;
   1:  PR[GP1:91,2] = PR[GP1:90,2] + 25.632;
   1:L PR[91] 10mm/sec CNT100;
   1:  PR[GP1:91,1] = PR[GP1:90,1] + -50.446;
   1:  PR[GP1:91,2] = PR[GP1:90,2] + 17.725;
   1:L PR[91] 10mm/sec CNT100;
   1:  PR[GP1:91,1] = PR[GP1:90,1] + -52.269;
   1:  PR[GP1:91,2] = PR[GP1:90,2] + 13.595;
   1:L PR[91] 10mm/sec CNT100;
   1:  PR[GP1:91,1] = PR[GP1:90,1] + -53.766;
   1:  PR[GP1:91,2] = PR[GP1:90,2] + 4.717;
   1:L PR[91] 10mm/sec CNT100;
   1:  PR[GP1:91,1] = PR[GP1:90,1] + -53.769;
   1:  PR[GP1:91,2] = PR[GP1:90,2] + 4.501;
   1:L PR[91] 10mm/sec CNT100;
   1:  PR[GP1:91,1] = PR[GP1:90,1] + -54.356;
   1:  PR[GP1:91,2] = PR[GP1:90,2] + 0.287;
   1:L PR[91] 10mm/sec CNT100;
   1:  PR[GP1:91,1] = PR[GP1:90,1] + -52.899;
   1:  PR[GP1:91,2] = PR[GP1:90,2] + -8.532;
   1:L PR[91] 10mm/sec CNT100;
   1:  PR[GP1:91,1] = PR[GP1:90,1] + -52.272;
   1:  PR[GP1:91,2] = PR[GP1:90,2] + -13.026;
   1:L PR[91] 10mm/sec CNT100;
   1:  PR[GP1:91,1] = PR[GP1:90,1] + -50.453;
   1:  PR[GP1:91,2] = PR[GP1:90,2] + -17.149;
   1:L PR[91] 10mm/sec CNT100;
   1:  PR[GP1:91,1] = PR[GP1:90,1] + -46.169;
   1:  PR[GP1:91,2] = PR[GP1:90,2] + -25.044;
   1:L PR[91] 10mm/sec CNT100;
   1:  PR[GP1:91,1] = PR[GP1:90,1] + -43.155;
   1:  PR[GP1:91,2] = PR[GP1:90,2] + -28.675;
   1:L PR[91] 10mm/sec CNT100;
   1:  PR[GP1:91,1] = PR[GP1:90,1] + -36.710;
   1:  PR[GP1:91,2] = PR[GP1:90,2] + -34.659;
   1:L PR[91] 10mm/sec CNT100;
   1:  PR[GP1:91,1] = PR[GP1:90,1] + -31.006;
   1:  PR[GP1:91,2] = PR[GP1:90,2] + -38.191;
   1:L PR[91] 10mm/sec CNT100;
   1:  PR[GP1:91,1] = PR[GP1:90,1] + -23.175;
   1:  PR[GP1:91,2] = PR[GP1:90,2] + -41.769;
   1:L PR[91] 10mm/sec CNT100;
   1:  PR[GP1:91,1] = PR[GP1:90,1] + -16.129;
   1:  PR[GP1:91,2] = PR[GP1:90,2] + -43.087;
   1:L PR[91] 10mm/sec CNT100;
   1:  PR[GP1:91,1] = PR[GP1:90,1] + -7.822;
   1:  PR[GP1:91,2] = PR[GP1:90,2] + -43.998;
   1:L PR[91] 10mm/sec CNT100;
   1:  PR[GP1:91,1] = PR[GP1:90,1] + -0.724;
   1:  PR[GP1:91,2] = PR[GP1:90,2] + -42.808;
   1:L PR[91] 10mm/sec CNT100;
   1:  PR[GP1:91,1] = PR[GP1:90,1] + -0.261;
   1:  PR[GP1:91,2] = PR[GP1:90,2] + -42.709;
   1:L PR[91] 10mm/sec CNT100;
   1:  PR[GP1:91,1] = PR[GP1:90,1] + 7.103;
   1:  PR[GP1:91,2] = PR[GP1:90,2] + -44.127;
   1:  PR[GP1:91,3] = PR[GP1:90,3] + 104.615;
   1:L PR[91] 10mm/sec CNT100;
   1:  PR[GP1:91,1] = PR[GP1:90,1] + 15.198;
   1:  PR[GP1:91,2] = PR[GP1:90,2] + -43.238;
   1:L PR[91] 10mm/sec CNT100;
   1:  PR[GP1:91,1] = PR[GP1:90,1] + 22.522;
   1:  PR[GP1:91,2] = PR[GP1:90,2] + -41.869;
   1:L PR[91] 10mm/sec CNT100;
   1:  PR[GP1:91,1] = PR[GP1:90,1] + 30.154;
   1:  PR[GP1:91,2] = PR[GP1:90,2] + -38.385;
   1:L PR[91] 10mm/sec CNT100;
   1:  PR[GP1:91,1] = PR[GP1:90,1] + 36.106;
   1:  PR[GP1:91,2] = PR[GP1:90,2] + -34.699;
   1:L PR[91] 10mm/sec CNT100;
   1:  PR[GP1:91,1] = PR[GP1:90,1] + 42.387;
   1:  PR[GP1:91,2] = PR[GP1:90,2] + -28.860;
   1:L PR[91] 10mm/sec CNT100;
   1:  PR[GP1:91,1] = PR[GP1:90,1] + 45.545;
   1:  PR[GP1:91,2] = PR[GP1:90,2] + -25.055;
   1:L PR[91] 10mm/sec CNT100;
   1:  PR[GP1:91,1] = PR[GP1:90,1] + 49.720;
   1:  PR[GP1:91,2] = PR[GP1:90,2] + -17.374;
   1:L PR[91] 10mm/sec CNT100;
   1:  PR[GP1:91,1] = PR[GP1:90,1] + 51.636;
   1:  PR[GP1:91,2] = PR[GP1:90,2] + -13.033;
   1:L PR[91] 10mm/sec CNT100;
   1:  PR[GP1:91,1] = PR[GP1:90,1] + 53.089;
   1:  PR[GP1:91,2] = PR[GP1:90,2] + -4.390;
   1:L PR[91] 10mm/sec CNT100;
   1:  PR[GP1:91,1] = PR[GP1:90,1] + 53.091;
   1:  PR[GP1:91,2] = PR[GP1:90,2] + -4.179;
   1:L PR[91] 10mm/sec CNT100;
   1:  PR[GP1:91,1] = PR[GP1:90,1] + 53.712;
   1:  PR[GP1:91,2] = PR[GP1:90,2] + 0.271;
   1:L PR[91] 10mm/sec CNT100;
   1:  PR[GP1:91,1] = PR[GP1:90,1] + 52.286;
   1:  PR[GP1:91,2] = PR[GP1:90,2] + 8.893;
   1:L PR[91] 10mm/sec CNT100;
   1:  PR[GP1:91,1] = PR[GP1:90,1] + 51.627;
   1:  PR[GP1:91,2] = PR[GP1:90,2] + 13.617;
   1:L PR[91] 10mm/sec CNT100;
   1:  PR[GP1:91,1] = PR[GP1:90,1] + 49.714;
   1:  PR[GP1:91,2] = PR[GP1:90,2] + 17.950;
   1:L PR[91] 10mm/sec CNT100;
   1:  PR[GP1:91,1] = PR[GP1:90,1] + 45.523;
   1:  PR[GP1:91,2] = PR[GP1:90,2] + 25.642;
   1:L PR[91] 10mm/sec CNT100;
   1:  PR[GP1:91,1] = PR[GP1:90,1] + 42.364;
   1:  PR[GP1:91,2] = PR[GP1:90,2] + 29.448;
   1:L PR[91] 10mm/sec CNT100;
   1:  PR[GP1:91,1] = PR[GP1:90,1] + 36.061;
   1:  PR[GP1:91,2] = PR[GP1:90,2] + 35.286;
   1:L PR[91] 10mm/sec CNT100;
   1:  PR[GP1:91,1] = PR[GP1:90,1] + 30.107;
   1:  PR[GP1:91,2] = PR[GP1:90,2] + 38.974;
   1:L PR[91] 10mm/sec CNT100;
   1:  PR[GP1:91,1] = PR[GP1:90,1] + 22.455;
   1:  PR[GP1:91,2] = PR[GP1:90,2] + 42.445;
   1:L PR[91] 10mm/sec CNT100;
   1:  PR[GP1:91,1] = PR[GP1:90,1] + 15.128;
   1:  PR[GP1:91,2] = PR[GP1:90,2] + 43.815;
   1:L PR[91] 10mm/sec CNT100;
   1:  PR[GP1:91,1] = PR[GP1:90,1] + 7.021;
   1:  PR[GP1:91,2] = PR[GP1:90,2] + 44.680;
   1:L PR[91] 10mm/sec CNT100;
   1:  PR[GP1:91,1] = PR[GP1:90,1] + -0.261;
   1:  PR[GP1:91,2] = PR[GP1:90,2] + 43.400;
   1:L PR[91] 10mm/sec CNT100;
   1:  PR[GP1:91,1] = PR[GP1:90,1] + -7.551;
   1:  PR[GP1:91,2] = PR[GP1:90,2] + 44.680;
   1:L PR[91] 10mm/sec CNT100;
   1:  PR[GP1:91,1] = PR[GP1:90,1] + -15.657;
   1:  PR[GP1:91,2] = PR[GP1:90,2] + 43.815;
   1:L PR[91] 10mm/sec CNT100;
   1:  PR[GP1:91,1] = PR[GP1:90,1] + -22.982;
   1:  PR[GP1:91,2] = PR[GP1:90,2] + 42.446;
   1:L PR[91] 10mm/sec CNT100;
   1:  PR[GP1:91,1] = PR[GP1:90,1] + -30.634;
   1:  PR[GP1:91,2] = PR[GP1:90,2] + 38.972;
   1:L PR[91] 10mm/sec CNT100;
   1:  PR[GP1:91,1] = PR[GP1:90,1] + -36.587;
   1:  PR[GP1:91,2] = PR[GP1:90,2] + 35.285;
   1:L PR[91] 10mm/sec CNT100;
   1:  PR[GP1:91,1] = PR[GP1:90,1] + -42.889;
   1:  PR[GP1:91,2] = PR[GP1:90,2] + 29.453;
   1:L PR[91] 10mm/sec CNT100;
   1:  PR[GP1:91,1] = PR[GP1:90,1] + -46.049;
   1:  PR[GP1:91,2] = PR[GP1:90,2] + 25.648;
   1:L PR[91] 10mm/sec CNT100;
   1:  PR[GP1:91,1] = PR[GP1:90,1] + -50.240;
   1:  PR[GP1:91,2] = PR[GP1:90,2] + 17.941;
   1:L PR[91] 10mm/sec CNT100;
   1:  PR[GP1:91,1] = PR[GP1:90,1] + -52.157;
   1:  PR[GP1:91,2] = PR[GP1:90,2] + 13.600;
   1:L PR[91] 10mm/sec CNT100;
   1:  PR[GP1:91,1] = PR[GP1:90,1] + -53.615;
   1:  PR[GP1:91,2] = PR[GP1:90,2] + 4.948;
   1:L PR[91] 10mm/sec CNT100;
   1:  PR[GP1:91,1] = PR[GP1:90,1] + -53.618;
   1:  PR[GP1:91,2] = PR[GP1:90,2] + 4.737;
   1:L PR[91] 10mm/sec CNT100;
   1:  PR[GP1:91,1] = PR[GP1:90,1] + -54.238;
   1:  PR[GP1:91,2] = PR[GP1:90,2] + 0.287;
   1:L PR[91] 10mm/sec CNT100;
   1:  PR[GP1:91,1] = PR[GP1:90,1] + -52.818;
   1:  PR[GP1:91,2] = PR[GP1:90,2] + -8.308;
   1:L PR[91] 10mm/sec CNT100;
   1:  PR[GP1:91,1] = PR[GP1:90,1] + -52.159;
   1:  PR[GP1:91,2] = PR[GP1:90,2] + -13.032;
   1:L PR[91] 10mm/sec CNT100;
   1:  PR[GP1:91,1] = PR[GP1:90,1] + -50.246;
   1:  PR[GP1:91,2] = PR[GP1:90,2] + -17.365;
   1:L PR[91] 10mm/sec CNT100;
   1:  PR[GP1:91,1] = PR[GP1:90,1] + -46.072;
   1:  PR[GP1:91,2] = PR[GP1:90,2] + -25.060;
   1:L PR[91] 10mm/sec CNT100;
   1:  PR[GP1:91,1] = PR[GP1:90,1] + -42.913;
   1:  PR[GP1:91,2] = PR[GP1:90,2] + -28.865;
   1:L PR[91] 10mm/sec CNT100;
   1:  PR[GP1:91,1] = PR[GP1:90,1] + -36.632;
   1:  PR[GP1:91,2] = PR[GP1:90,2] + -34.697;
   1:L PR[91] 10mm/sec CNT100;
   1:  PR[GP1:91,1] = PR[GP1:90,1] + -30.681;
   1:  PR[GP1:91,2] = PR[GP1:90,2] + -38.383;
   1:L PR[91] 10mm/sec CNT100;
   1:  PR[GP1:91,1] = PR[GP1:90,1] + -23.049;
   1:  PR[GP1:91,2] = PR[GP1:90,2] + -41.869;
   1:L PR[91] 10mm/sec CNT100;
   1:  PR[GP1:91,1] = PR[GP1:90,1] + -15.728;
   1:  PR[GP1:91,2] = PR[GP1:90,2] + -43.238;
   1:L PR[91] 10mm/sec CNT100;
   1:  PR[GP1:91,1] = PR[GP1:90,1] + -7.633;
   1:  PR[GP1:91,2] = PR[GP1:90,2] + -44.127;
   1:L PR[91] 10mm/sec CNT100;
   1:  PR[GP1:91,1] = PR[GP1:90,1] + -0.261;
   1:  PR[GP1:91,2] = PR[GP1:90,2] + -42.891;
   1:L PR[91] 10mm/sec CNT100;
   1:  PR[GP1:91,1] = PR[GP1:90,1] + 6.914;
   1:  PR[GP1:91,2] = PR[GP1:90,2] + -44.255;
   1:  PR[GP1:91,3] = PR[GP1:90,3] + 105.225;
   1:L PR[91] 10mm/sec CNT100;
   1:  PR[GP1:91,1] = PR[GP1:90,1] + 14.798;
   1:  PR[GP1:91,2] = PR[GP1:90,2] + -43.389;
   1:L PR[91] 10mm/sec CNT100;
   1:  PR[GP1:91,1] = PR[GP1:90,1] + 22.395;
   1:  PR[GP1:91,2] = PR[GP1:90,2] + -41.969;
   1:L PR[91] 10mm/sec CNT100;
   1:  PR[GP1:91,1] = PR[GP1:90,1] + 29.828;
   1:  PR[GP1:91,2] = PR[GP1:90,2] + -38.576;
   1:L PR[91] 10mm/sec CNT100;
   1:  PR[GP1:91,1] = PR[GP1:90,1] + 36.027;
   1:  PR[GP1:91,2] = PR[GP1:90,2] + -34.737;
   1:L PR[91] 10mm/sec CNT100;
   1:  PR[GP1:91,1] = PR[GP1:90,1] + 42.145;
   1:  PR[GP1:91,2] = PR[GP1:90,2] + -29.050;
   1:L PR[91] 10mm/sec CNT100;
   1:  PR[GP1:91,1] = PR[GP1:90,1] + 45.448;
   1:  PR[GP1:91,2] = PR[GP1:90,2] + -25.072;
   1:L PR[91] 10mm/sec CNT100;
   1:  PR[GP1:91,1] = PR[GP1:90,1] + 49.514;
   1:  PR[GP1:91,2] = PR[GP1:90,2] + -17.590;
   1:L PR[91] 10mm/sec CNT100;
   1:  PR[GP1:91,1] = PR[GP1:90,1] + 51.523;
   1:  PR[GP1:91,2] = PR[GP1:90,2] + -13.038;
   1:L PR[91] 10mm/sec CNT100;
   1:  PR[GP1:91,1] = PR[GP1:90,1] + 52.938;
   1:  PR[GP1:91,2] = PR[GP1:90,2] + -4.620;
   1:L PR[91] 10mm/sec CNT100;
   1:  PR[GP1:91,1] = PR[GP1:90,1] + 52.941;
   1:  PR[GP1:91,2] = PR[GP1:90,2] + -4.415;
   1:L PR[91] 10mm/sec CNT100;
   1:  PR[GP1:91,1] = PR[GP1:90,1] + 53.594;
   1:  PR[GP1:91,2] = PR[GP1:90,2] + 0.271;
   1:L PR[91] 10mm/sec CNT100;
   1:  PR[GP1:91,1] = PR[GP1:90,1] + 52.205;
   1:  PR[GP1:91,2] = PR[GP1:90,2] + 8.669;
   1:L PR[91] 10mm/sec CNT100;
   1:  PR[GP1:91,1] = PR[GP1:90,1] + 51.514;
   1:  PR[GP1:91,2] = PR[GP1:90,2] + 13.621;
   1:L PR[91] 10mm/sec CNT100;
   1:  PR[GP1:91,1] = PR[GP1:90,1] + 49.508;
   1:  PR[GP1:91,2] = PR[GP1:90,2] + 18.165;
   1:L PR[91] 10mm/sec CNT100;
   1:  PR[GP1:91,1] = PR[GP1:90,1] + 45.426;
   1:  PR[GP1:91,2] = PR[GP1:90,2] + 25.658;
   1:L PR[91] 10mm/sec CNT100;
   1:  PR[GP1:91,1] = PR[GP1:90,1] + 42.122;
   1:  PR[GP1:91,2] = PR[GP1:90,2] + 29.637;
   1:L PR[91] 10mm/sec CNT100;
   1:  PR[GP1:91,1] = PR[GP1:90,1] + 35.984;
   1:  PR[GP1:91,2] = PR[GP1:90,2] + 35.324;
   1:L PR[91] 10mm/sec CNT100;
   1:  PR[GP1:91,1] = PR[GP1:90,1] + 29.782;
   1:  PR[GP1:91,2] = PR[GP1:90,2] + 39.164;
   1:L PR[91] 10mm/sec CNT100;
   1:  PR[GP1:91,1] = PR[GP1:90,1] + 22.330;
   1:  PR[GP1:91,2] = PR[GP1:90,2] + 42.545;
   1:L PR[91] 10mm/sec CNT100;
   1:  PR[GP1:91,1] = PR[GP1:90,1] + 14.729;
   1:  PR[GP1:91,2] = PR[GP1:90,2] + 43.966;
   1:L PR[91] 10mm/sec CNT100;
   1:  PR[GP1:91,1] = PR[GP1:90,1] + 6.834;
   1:  PR[GP1:91,2] = PR[GP1:90,2] + 44.809;
   1:L PR[91] 10mm/sec CNT100;
   1:  PR[GP1:91,1] = PR[GP1:90,1] + -0.261;
   1:  PR[GP1:91,2] = PR[GP1:90,2] + 43.561;
   1:L PR[91] 10mm/sec CNT100;
   1:  PR[GP1:91,1] = PR[GP1:90,1] + -7.364;
   1:  PR[GP1:91,2] = PR[GP1:90,2] + 44.809;
   1:L PR[91] 10mm/sec CNT100;
   1:  PR[GP1:91,1] = PR[GP1:90,1] + -15.259;
   1:  PR[GP1:91,2] = PR[GP1:90,2] + 43.967;
   1:L PR[91] 10mm/sec CNT100;
   1:  PR[GP1:91,1] = PR[GP1:90,1] + -22.857;
   1:  PR[GP1:91,2] = PR[GP1:90,2] + 42.545;
   1:L PR[91] 10mm/sec CNT100;
   1:  PR[GP1:91,1] = PR[GP1:90,1] + -30.310;
   1:  PR[GP1:91,2] = PR[GP1:90,2] + 39.162;
   1:L PR[91] 10mm/sec CNT100;
   1:  PR[GP1:91,1] = PR[GP1:90,1] + -36.510;
   1:  PR[GP1:91,2] = PR[GP1:90,2] + 35.322;
   1:L PR[91] 10mm/sec CNT100;
   1:  PR[GP1:91,1] = PR[GP1:90,1] + -42.648;
   1:  PR[GP1:91,2] = PR[GP1:90,2] + 29.643;
   1:L PR[91] 10mm/sec CNT100;
   1:  PR[GP1:91,1] = PR[GP1:90,1] + -45.952;
   1:  PR[GP1:91,2] = PR[GP1:90,2] + 25.664;
   1:L PR[91] 10mm/sec CNT100;
   1:  PR[GP1:91,1] = PR[GP1:90,1] + -50.034;
   1:  PR[GP1:91,2] = PR[GP1:90,2] + 18.157;
   1:L PR[91] 10mm/sec CNT100;
   1:  PR[GP1:91,1] = PR[GP1:90,1] + -52.044;
   1:  PR[GP1:91,2] = PR[GP1:90,2] + 13.605;
   1:L PR[91] 10mm/sec CNT100;
   1:  PR[GP1:91,1] = PR[GP1:90,1] + -53.465;
   1:  PR[GP1:91,2] = PR[GP1:90,2] + 5.178;
   1:L PR[91] 10mm/sec CNT100;
   1:  PR[GP1:91,1] = PR[GP1:90,1] + -53.467;
   1:  PR[GP1:91,2] = PR[GP1:90,2] + 4.973;
   1:L PR[91] 10mm/sec CNT100;
   1:  PR[GP1:91,1] = PR[GP1:90,1] + -54.120;
   1:  PR[GP1:91,2] = PR[GP1:90,2] + 0.287;
   1:L PR[91] 10mm/sec CNT100;
   1:  PR[GP1:91,1] = PR[GP1:90,1] + -52.737;
   1:  PR[GP1:91,2] = PR[GP1:90,2] + -8.085;
   1:L PR[91] 10mm/sec CNT100;
   1:  PR[GP1:91,1] = PR[GP1:90,1] + -52.046;
   1:  PR[GP1:91,2] = PR[GP1:90,2] + -13.037;
   1:L PR[91] 10mm/sec CNT100;
   1:  PR[GP1:91,1] = PR[GP1:90,1] + -50.040;
   1:  PR[GP1:91,2] = PR[GP1:90,2] + -17.582;
   1:L PR[91] 10mm/sec CNT100;
   1:  PR[GP1:91,1] = PR[GP1:90,1] + -45.974;
   1:  PR[GP1:91,2] = PR[GP1:90,2] + -25.077;
   1:L PR[91] 10mm/sec CNT100;
   1:  PR[GP1:91,1] = PR[GP1:90,1] + -42.671;
   1:  PR[GP1:91,2] = PR[GP1:90,2] + -29.055;
   1:L PR[91] 10mm/sec CNT100;
   1:  PR[GP1:91,1] = PR[GP1:90,1] + -36.553;
   1:  PR[GP1:91,2] = PR[GP1:90,2] + -34.735;
   1:L PR[91] 10mm/sec CNT100;
   1:  PR[GP1:91,1] = PR[GP1:90,1] + -30.356;
   1:  PR[GP1:91,2] = PR[GP1:90,2] + -38.574;
   1:L PR[91] 10mm/sec CNT100;
   1:  PR[GP1:91,1] = PR[GP1:90,1] + -22.923;
   1:  PR[GP1:91,2] = PR[GP1:90,2] + -41.969;
   1:L PR[91] 10mm/sec CNT100;
   1:  PR[GP1:91,1] = PR[GP1:90,1] + -15.328;
   1:  PR[GP1:91,2] = PR[GP1:90,2] + -43.390;
   1:L PR[91] 10mm/sec CNT100;
   1:  PR[GP1:91,1] = PR[GP1:90,1] + -7.444;
   1:  PR[GP1:91,2] = PR[GP1:90,2] + -44.255;
   1:L PR[91] 10mm/sec CNT100;
   1:  PR[GP1:91,1] = PR[GP1:90,1] + -0.261;
   1:  PR[GP1:91,2] = PR[GP1:90,2] + -43.051;
   1:L PR[91] 10mm/sec CNT100;
   1:  PR[GP1:91,1] = PR[GP1:90,1] + 6.724;
   1:  PR[GP1:91,2] = PR[GP1:90,2] + -44.384;
   1:  PR[GP1:91,3] = PR[GP1:90,3] + 105.835;
   1:L PR[91] 10mm/sec CNT100;
   1:  PR[GP1:91,1] = PR[GP1:90,1] + 14.397;
   1:  PR[GP1:91,2] = PR[GP1:90,2] + -43.541;
   1:L PR[91] 10mm/sec CNT100;
   1:  PR[GP1:91,1] = PR[GP1:90,1] + 22.269;
   1:  PR[GP1:91,2] = PR[GP1:90,2] + -42.070;
   1:L PR[91] 10mm/sec CNT100;
   1:  PR[GP1:91,1] = PR[GP1:90,1] + 29.503;
   1:  PR[GP1:91,2] = PR[GP1:90,2] + -38.768;
   1:L PR[91] 10mm/sec CNT100;
   1:  PR[GP1:91,1] = PR[GP1:90,1] + 35.949;
   1:  PR[GP1:91,2] = PR[GP1:90,2] + -34.775;
   1:L PR[91] 10mm/sec CNT100;
   1:  PR[GP1:91,1] = PR[GP1:90,1] + 41.903;
   1:  PR[GP1:91,2] = PR[GP1:90,2] + -29.240;
   1:L PR[91] 10mm/sec CNT100;
   1:  PR[GP1:91,1] = PR[GP1:90,1] + 45.350;
   1:  PR[GP1:91,2] = PR[GP1:90,2] + -25.088;
   1:L PR[91] 10mm/sec CNT100;
   1:  PR[GP1:91,1] = PR[GP1:90,1] + 49.308;
   1:  PR[GP1:91,2] = PR[GP1:90,2] + -17.806;
   1:L PR[91] 10mm/sec CNT100;
   1:  PR[GP1:91,1] = PR[GP1:90,1] + 51.410;
   1:  PR[GP1:91,2] = PR[GP1:90,2] + -13.043;
   1:L PR[91] 10mm/sec CNT100;
   1:  PR[GP1:91,1] = PR[GP1:90,1] + 52.787;
   1:  PR[GP1:91,2] = PR[GP1:90,2] + -4.851;
   1:L PR[91] 10mm/sec CNT100;
   1:  PR[GP1:91,1] = PR[GP1:90,1] + 52.790;
   1:  PR[GP1:91,2] = PR[GP1:90,2] + -4.651;
   1:L PR[91] 10mm/sec CNT100;
   1:  PR[GP1:91,1] = PR[GP1:90,1] + 53.476;
   1:  PR[GP1:91,2] = PR[GP1:90,2] + 0.271;
   1:L PR[91] 10mm/sec CNT100;
   1:  PR[GP1:91,1] = PR[GP1:90,1] + 52.124;
   1:  PR[GP1:91,2] = PR[GP1:90,2] + 8.445;
   1:L PR[91] 10mm/sec CNT100;
   1:  PR[GP1:91,1] = PR[GP1:90,1] + 51.401;
   1:  PR[GP1:91,2] = PR[GP1:90,2] + 13.626;
   1:L PR[91] 10mm/sec CNT100;
   1:  PR[GP1:91,1] = PR[GP1:90,1] + 49.302;
   1:  PR[GP1:91,2] = PR[GP1:90,2] + 18.381;
   1:L PR[91] 10mm/sec CNT100;
   1:  PR[GP1:91,1] = PR[GP1:90,1] + 45.328;
   1:  PR[GP1:91,2] = PR[GP1:90,2] + 25.674;
   1:L PR[91] 10mm/sec CNT100;
   1:  PR[GP1:91,1] = PR[GP1:90,1] + 41.881;
   1:  PR[GP1:91,2] = PR[GP1:90,2] + 29.827;
   1:L PR[91] 10mm/sec CNT100;
   1:  PR[GP1:91,1] = PR[GP1:90,1] + 35.907;
   1:  PR[GP1:91,2] = PR[GP1:90,2] + 35.361;
   1:L PR[91] 10mm/sec CNT100;
   1:  PR[GP1:91,1] = PR[GP1:90,1] + 29.458;
   1:  PR[GP1:91,2] = PR[GP1:90,2] + 39.355;
   1:L PR[91] 10mm/sec CNT100;
   1:  PR[GP1:91,1] = PR[GP1:90,1] + 22.206;
   1:  PR[GP1:91,2] = PR[GP1:90,2] + 42.645;
   1:L PR[91] 10mm/sec CNT100;
   1:  PR[GP1:91,1] = PR[GP1:90,1] + 14.330;
   1:  PR[GP1:91,2] = PR[GP1:90,2] + 44.117;
   1:L PR[91] 10mm/sec CNT100;
   1:  PR[GP1:91,1] = PR[GP1:90,1] + 6.647;
   1:  PR[GP1:91,2] = PR[GP1:90,2] + 44.938;
   1:L PR[91] 10mm/sec CNT100;
   1:  PR[GP1:91,1] = PR[GP1:90,1] + -0.261;
   1:  PR[GP1:91,2] = PR[GP1:90,2] + 43.723;
   1:L PR[91] 10mm/sec CNT100;
   1:  PR[GP1:91,1] = PR[GP1:90,1] + -7.177;
   1:  PR[GP1:91,2] = PR[GP1:90,2] + 44.937;
   1:L PR[91] 10mm/sec CNT100;
   1:  PR[GP1:91,1] = PR[GP1:90,1] + -14.860;
   1:  PR[GP1:91,2] = PR[GP1:90,2] + 44.118;
   1:L PR[91] 10mm/sec CNT100;
   1:  PR[GP1:91,1] = PR[GP1:90,1] + -22.733;
   1:  PR[GP1:91,2] = PR[GP1:90,2] + 42.645;
   1:L PR[91] 10mm/sec CNT100;
   1:  PR[GP1:91,1] = PR[GP1:90,1] + -29.986;
   1:  PR[GP1:91,2] = PR[GP1:90,2] + 39.353;
   1:L PR[91] 10mm/sec CNT100;
   1:  PR[GP1:91,1] = PR[GP1:90,1] + -36.432;
   1:  PR[GP1:91,2] = PR[GP1:90,2] + 35.360;
   1:L PR[91] 10mm/sec CNT100;
   1:  PR[GP1:91,1] = PR[GP1:90,1] + -42.407;
   1:  PR[GP1:91,2] = PR[GP1:90,2] + 29.832;
   1:L PR[91] 10mm/sec CNT100;
   1:  PR[GP1:91,1] = PR[GP1:90,1] + -45.854;
   1:  PR[GP1:91,2] = PR[GP1:90,2] + 25.679;
   1:L PR[91] 10mm/sec CNT100;
   1:  PR[GP1:91,1] = PR[GP1:90,1] + -49.828;
   1:  PR[GP1:91,2] = PR[GP1:90,2] + 18.373;
   1:L PR[91] 10mm/sec CNT100;
   1:  PR[GP1:91,1] = PR[GP1:90,1] + -51.931;
   1:  PR[GP1:91,2] = PR[GP1:90,2] + 13.609;
   1:L PR[91] 10mm/sec CNT100;
   1:  PR[GP1:91,1] = PR[GP1:90,1] + -53.314;
   1:  PR[GP1:91,2] = PR[GP1:90,2] + 5.409;
   1:L PR[91] 10mm/sec CNT100;
   1:  PR[GP1:91,1] = PR[GP1:90,1] + -53.316;
   1:  PR[GP1:91,2] = PR[GP1:90,2] + 5.210;
   1:L PR[91] 10mm/sec CNT100;
   1:  PR[GP1:91,1] = PR[GP1:90,1] + -54.003;
   1:  PR[GP1:91,2] = PR[GP1:90,2] + 0.287;
   1:L PR[91] 10mm/sec CNT100;
   1:  PR[GP1:91,1] = PR[GP1:90,1] + -52.656;
   1:  PR[GP1:91,2] = PR[GP1:90,2] + -7.861;
   1:L PR[91] 10mm/sec CNT100;
   1:  PR[GP1:91,1] = PR[GP1:90,1] + -51.933;
   1:  PR[GP1:91,2] = PR[GP1:90,2] + -13.042;
   1:L PR[91] 10mm/sec CNT100;
   1:  PR[GP1:91,1] = PR[GP1:90,1] + -49.834;
   1:  PR[GP1:91,2] = PR[GP1:90,2] + -17.798;
   1:L PR[91] 10mm/sec CNT100;
   1:  PR[GP1:91,1] = PR[GP1:90,1] + -45.876;
   1:  PR[GP1:91,2] = PR[GP1:90,2] + -25.093;
   1:L PR[91] 10mm/sec CNT100;
   1:  PR[GP1:91,1] = PR[GP1:90,1] + -42.429;
   1:  PR[GP1:91,2] = PR[GP1:90,2] + -29.246;
   1:L PR[91] 10mm/sec CNT100;
   1:  PR[GP1:91,1] = PR[GP1:90,1] + -36.475;
   1:  PR[GP1:91,2] = PR[GP1:90,2] + -34.774;
   1:L PR[91] 10mm/sec CNT100;
   1:  PR[GP1:91,1] = PR[GP1:90,1] + -30.030;
   1:  PR[GP1:91,2] = PR[GP1:90,2] + -38.765;
   1:L PR[91] 10mm/sec CNT100;
   1:  PR[GP1:91,1] = PR[GP1:90,1] + -22.797;
   1:  PR[GP1:91,2] = PR[GP1:90,2] + -42.070;
   1:L PR[91] 10mm/sec CNT100;
   1:  PR[GP1:91,1] = PR[GP1:90,1] + -14.928;
   1:  PR[GP1:91,2] = PR[GP1:90,2] + -43.542;
   1:L PR[91] 10mm/sec CNT100;
   1:  PR[GP1:91,1] = PR[GP1:90,1] + -7.254;
   1:  PR[GP1:91,2] = PR[GP1:90,2] + -44.384;
   1:L PR[91] 10mm/sec CNT100;
   1:  PR[GP1:91,1] = PR[GP1:90,1] + -0.261;
   1:  PR[GP1:91,2] = PR[GP1:90,2] + -43.211;
   1:L PR[91] 10mm/sec CNT100;
   1:  PR[GP1:91,1] = PR[GP1:90,1] + 6.535;
   1:  PR[GP1:91,2] = PR[GP1:90,2] + -44.512;
   1:  PR[GP1:91,3] = PR[GP1:90,3] + 106.445;
   1:L PR[91] 10mm/sec CNT100;
   1:  PR[GP1:91,1] = PR[GP1:90,1] + 13.997;
   1:  PR[GP1:91,2] = PR[GP1:90,2] + -43.693;
   1:L PR[91] 10mm/sec CNT100;
   1:  PR[GP1:91,1] = PR[GP1:90,1] + 22.143;
   1:  PR[GP1:91,2] = PR[GP1:90,2] + -42.170;
   1:L PR[91] 10mm/sec CNT100;
   1:  PR[GP1:91,1] = PR[GP1:90,1] + 29.177;
   1:  PR[GP1:91,2] = PR[GP1:90,2] + -38.959;
   1:L PR[91] 10mm/sec CNT100;
   1:  PR[GP1:91,1] = PR[GP1:90,1] + 35.871;
   1:  PR[GP1:91,2] = PR[GP1:90,2] + -34.813;
   1:L PR[91] 10mm/sec CNT100;
   1:  PR[GP1:91,1] = PR[GP1:90,1] + 41.661;
   1:  PR[GP1:91,2] = PR[GP1:90,2] + -29.431;
   1:L PR[91] 10mm/sec CNT100;
   1:  PR[GP1:91,1] = PR[GP1:90,1] + 45.252;
   1:  PR[GP1:91,2] = PR[GP1:90,2] + -25.105;
   1:L PR[91] 10mm/sec CNT100;
   1:  PR[GP1:91,1] = PR[GP1:90,1] + 49.102;
   1:  PR[GP1:91,2] = PR[GP1:90,2] + -18.023;
   1:L PR[91] 10mm/sec CNT100;
   1:  PR[GP1:91,1] = PR[GP1:90,1] + 51.298;
   1:  PR[GP1:91,2] = PR[GP1:90,2] + -13.048;
   1:L PR[91] 10mm/sec CNT100;
   1:  PR[GP1:91,1] = PR[GP1:90,1] + 52.636;
   1:  PR[GP1:91,2] = PR[GP1:90,2] + -5.082;
   1:L PR[91] 10mm/sec CNT100;
   1:  PR[GP1:91,1] = PR[GP1:90,1] + 52.639;
   1:  PR[GP1:91,2] = PR[GP1:90,2] + -4.888;
   1:L PR[91] 10mm/sec CNT100;
   1:  PR[GP1:91,1] = PR[GP1:90,1] + 53.358;
   1:  PR[GP1:91,2] = PR[GP1:90,2] + 0.271;
   1:L PR[91] 10mm/sec CNT100;
   1:  PR[GP1:91,1] = PR[GP1:90,1] + 52.043;
   1:  PR[GP1:91,2] = PR[GP1:90,2] + 8.221;
   1:L PR[91] 10mm/sec CNT100;
   1:  PR[GP1:91,1] = PR[GP1:90,1] + 51.288;
   1:  PR[GP1:91,2] = PR[GP1:90,2] + 13.630;
   1:L PR[91] 10mm/sec CNT100;
   1:  PR[GP1:91,1] = PR[GP1:90,1] + 49.096;
   1:  PR[GP1:91,2] = PR[GP1:90,2] + 18.597;
   1:L PR[91] 10mm/sec CNT100;
   1:  PR[GP1:91,1] = PR[GP1:90,1] + 45.231;
   1:  PR[GP1:91,2] = PR[GP1:90,2] + 25.690;
   1:L PR[91] 10mm/sec CNT100;
   1:  PR[GP1:91,1] = PR[GP1:90,1] + 41.640;
   1:  PR[GP1:91,2] = PR[GP1:90,2] + 30.016;
   1:L PR[91] 10mm/sec CNT100;
   1:  PR[GP1:91,1] = PR[GP1:90,1] + 35.829;
   1:  PR[GP1:91,2] = PR[GP1:90,2] + 35.399;
   1:L PR[91] 10mm/sec CNT100;
   1:  PR[GP1:91,1] = PR[GP1:90,1] + 29.134;
   1:  PR[GP1:91,2] = PR[GP1:90,2] + 39.545;
   1:L PR[91] 10mm/sec CNT100;
   1:  PR[GP1:91,1] = PR[GP1:90,1] + 22.081;
   1:  PR[GP1:91,2] = PR[GP1:90,2] + 42.745;
   1:L PR[91] 10mm/sec CNT100;
   1:  PR[GP1:91,1] = PR[GP1:90,1] + 13.932;
   1:  PR[GP1:91,2] = PR[GP1:90,2] + 44.268;
   1:L PR[91] 10mm/sec CNT100;
   1:  PR[GP1:91,1] = PR[GP1:90,1] + 6.460;
   1:  PR[GP1:91,2] = PR[GP1:90,2] + 45.066;
   1:L PR[91] 10mm/sec CNT100;
   1:  PR[GP1:91,1] = PR[GP1:90,1] + -0.261;
   1:  PR[GP1:91,2] = PR[GP1:90,2] + 43.884;
   1:L PR[91] 10mm/sec CNT100;
   1:  PR[GP1:91,1] = PR[GP1:90,1] + -6.990;
   1:  PR[GP1:91,2] = PR[GP1:90,2] + 45.066;
   1:L PR[91] 10mm/sec CNT100;
   1:  PR[GP1:91,1] = PR[GP1:90,1] + -14.462;
   1:  PR[GP1:91,2] = PR[GP1:90,2] + 44.269;
   1:L PR[91] 10mm/sec CNT100;
   1:  PR[GP1:91,1] = PR[GP1:90,1] + -22.608;
   1:  PR[GP1:91,2] = PR[GP1:90,2] + 42.745;
   1:L PR[91] 10mm/sec CNT100;
   1:  PR[GP1:91,1] = PR[GP1:90,1] + -29.662;
   1:  PR[GP1:91,2] = PR[GP1:90,2] + 39.543;
   1:L PR[91] 10mm/sec CNT100;
   1:  PR[GP1:91,1] = PR[GP1:90,1] + -36.355;
   1:  PR[GP1:91,2] = PR[GP1:90,2] + 35.398;
   1:L PR[91] 10mm/sec CNT100;
   1:  PR[GP1:91,1] = PR[GP1:90,1] + -42.165;
   1:  PR[GP1:91,2] = PR[GP1:90,2] + 30.022;
   1:L PR[91] 10mm/sec CNT100;
   1:  PR[GP1:91,1] = PR[GP1:90,1] + -45.757;
   1:  PR[GP1:91,2] = PR[GP1:90,2] + 25.695;
   1:L PR[91] 10mm/sec CNT100;
   1:  PR[GP1:91,1] = PR[GP1:90,1] + -49.622;
   1:  PR[GP1:91,2] = PR[GP1:90,2] + 18.589;
   1:L PR[91] 10mm/sec CNT100;
   1:  PR[GP1:91,1] = PR[GP1:90,1] + -51.818;
   1:  PR[GP1:91,2] = PR[GP1:90,2] + 13.614;
   1:L PR[91] 10mm/sec CNT100;
   1:  PR[GP1:91,1] = PR[GP1:90,1] + -53.163;
   1:  PR[GP1:91,2] = PR[GP1:90,2] + 5.640;
   1:L PR[91] 10mm/sec CNT100;
   1:  PR[GP1:91,1] = PR[GP1:90,1] + -53.165;
   1:  PR[GP1:91,2] = PR[GP1:90,2] + 5.446;
   1:L PR[91] 10mm/sec CNT100;
   1:  PR[GP1:91,1] = PR[GP1:90,1] + -53.885;
   1:  PR[GP1:91,2] = PR[GP1:90,2] + 0.287;
   1:L PR[91] 10mm/sec CNT100;
   1:  PR[GP1:91,1] = PR[GP1:90,1] + -52.575;
   1:  PR[GP1:91,2] = PR[GP1:90,2] + -7.638;
   1:L PR[91] 10mm/sec CNT100;
   1:  PR[GP1:91,1] = PR[GP1:90,1] + -51.820;
   1:  PR[GP1:91,2] = PR[GP1:90,2] + -13.048;
   1:L PR[91] 10mm/sec CNT100;
   1:  PR[GP1:91,1] = PR[GP1:90,1] + -49.628;
   1:  PR[GP1:91,2] = PR[GP1:90,2] + -18.015;
   1:L PR[91] 10mm/sec CNT100;
   1:  PR[GP1:91,1] = PR[GP1:90,1] + -45.778;
   1:  PR[GP1:91,2] = PR[GP1:90,2] + -25.110;
   1:L PR[91] 10mm/sec CNT100;
   1:  PR[GP1:91,1] = PR[GP1:90,1] + -42.187;
   1:  PR[GP1:91,2] = PR[GP1:90,2] + -29.436;
   1:L PR[91] 10mm/sec CNT100;
   1:  PR[GP1:91,1] = PR[GP1:90,1] + -36.397;
   1:  PR[GP1:91,2] = PR[GP1:90,2] + -34.812;
   1:L PR[91] 10mm/sec CNT100;
   1:  PR[GP1:91,1] = PR[GP1:90,1] + -29.705;
   1:  PR[GP1:91,2] = PR[GP1:90,2] + -38.957;
   1:L PR[91] 10mm/sec CNT100;
   1:  PR[GP1:91,1] = PR[GP1:90,1] + -22.671;
   1:  PR[GP1:91,2] = PR[GP1:90,2] + -42.170;
   1:L PR[91] 10mm/sec CNT100;
   1:  PR[GP1:91,1] = PR[GP1:90,1] + -14.527;
   1:  PR[GP1:91,2] = PR[GP1:90,2] + -43.693;
   1:L PR[91] 10mm/sec CNT100;
   1:  PR[GP1:91,1] = PR[GP1:90,1] + -7.065;
   1:  PR[GP1:91,2] = PR[GP1:90,2] + -44.512;
   1:L PR[91] 10mm/sec CNT100;
   1:  PR[GP1:91,1] = PR[GP1:90,1] + -0.261;
   1:  PR[GP1:91,2] = PR[GP1:90,2] + -43.371;
   1:L PR[91] 10mm/sec CNT100;
   1:  PR[GP1:91,1] = PR[GP1:90,1] + 6.346;
   1:  PR[GP1:91,2] = PR[GP1:90,2] + -44.641;
   1:  PR[GP1:91,3] = PR[GP1:90,3] + 107.055;
   1:L PR[91] 10mm/sec CNT100;
   1:  PR[GP1:91,1] = PR[GP1:90,1] + 13.596;
   1:  PR[GP1:91,2] = PR[GP1:90,2] + -43.844;
   1:L PR[91] 10mm/sec CNT100;
   1:  PR[GP1:91,1] = PR[GP1:90,1] + 22.017;
   1:  PR[GP1:91,2] = PR[GP1:90,2] + -42.270;
   1:L PR[91] 10mm/sec CNT100;
   1:  PR[GP1:91,1] = PR[GP1:90,1] + 28.852;
   1:  PR[GP1:91,2] = PR[GP1:90,2] + -39.150;
   1:L PR[91] 10mm/sec CNT100;
   1:  PR[GP1:91,1] = PR[GP1:90,1] + 35.792;
   1:  PR[GP1:91,2] = PR[GP1:90,2] + -34.852;
   1:L PR[91] 10mm/sec CNT100;
   1:  PR[GP1:91,1] = PR[GP1:90,1] + 41.419;
   1:  PR[GP1:91,2] = PR[GP1:90,2] + -29.621;
   1:L PR[91] 10mm/sec CNT100;
   1:  PR[GP1:91,1] = PR[GP1:90,1] + 45.155;
   1:  PR[GP1:91,2] = PR[GP1:90,2] + -25.121;
   1:L PR[91] 10mm/sec CNT100;
   1:  PR[GP1:91,1] = PR[GP1:90,1] + 48.895;
   1:  PR[GP1:91,2] = PR[GP1:90,2] + -18.239;
   1:L PR[91] 10mm/sec CNT100;
   1:  PR[GP1:91,1] = PR[GP1:90,1] + 51.185;
   1:  PR[GP1:91,2] = PR[GP1:90,2] + -13.053;
   1:L PR[91] 10mm/sec CNT100;
   1:  PR[GP1:91,1] = PR[GP1:90,1] + 52.486;
   1:  PR[GP1:91,2] = PR[GP1:90,2] + -5.312;
   1:L PR[91] 10mm/sec CNT100;
   1:  PR[GP1:91,1] = PR[GP1:90,1] + 52.488;
   1:  PR[GP1:91,2] = PR[GP1:90,2] + -5.124;
   1:L PR[91] 10mm/sec CNT100;
   1:  PR[GP1:91,1] = PR[GP1:90,1] + 53.240;
   1:  PR[GP1:91,2] = PR[GP1:90,2] + 0.271;
   1:L PR[91] 10mm/sec CNT100;
   1:  PR[GP1:91,1] = PR[GP1:90,1] + 51.962;
   1:  PR[GP1:91,2] = PR[GP1:90,2] + 7.997;
   1:L PR[91] 10mm/sec CNT100;
   1:  PR[GP1:91,1] = PR[GP1:90,1] + 51.176;
   1:  PR[GP1:91,2] = PR[GP1:90,2] + 13.635;
   1:L PR[91] 10mm/sec CNT100;
   1:  PR[GP1:91,1] = PR[GP1:90,1] + 48.890;
   1:  PR[GP1:91,2] = PR[GP1:90,2] + 18.813;
   1:L PR[91] 10mm/sec CNT100;
   1:  PR[GP1:91,1] = PR[GP1:90,1] + 45.134;
   1:  PR[GP1:91,2] = PR[GP1:90,2] + 25.706;
   1:L PR[91] 10mm/sec CNT100;
   1:  PR[GP1:91,1] = PR[GP1:90,1] + 41.398;
   1:  PR[GP1:91,2] = PR[GP1:90,2] + 30.206;
   1:L PR[91] 10mm/sec CNT100;
   1:  PR[GP1:91,1] = PR[GP1:90,1] + 35.752;
   1:  PR[GP1:91,2] = PR[GP1:90,2] + 35.436;
   1:L PR[91] 10mm/sec CNT100;
   1:  PR[GP1:91,1] = PR[GP1:90,1] + 28.810;
   1:  PR[GP1:91,2] = PR[GP1:90,2] + 39.736;
   1:L PR[91] 10mm/sec CNT100;
   1:  PR[GP1:91,1] = PR[GP1:90,1] + 21.957;
   1:  PR[GP1:91,2] = PR[GP1:90,2] + 42.845;
   1:L PR[91] 10mm/sec CNT100;
   1:  PR[GP1:91,1] = PR[GP1:90,1] + 13.533;
   1:  PR[GP1:91,2] = PR[GP1:90,2] + 44.419;
   1:L PR[91] 10mm/sec CNT100;
   1:  PR[GP1:91,1] = PR[GP1:90,1] + 6.273;
   1:  PR[GP1:91,2] = PR[GP1:90,2] + 45.195;
   1:L PR[91] 10mm/sec CNT100;
   1:  PR[GP1:91,1] = PR[GP1:90,1] + -0.261;
   1:  PR[GP1:91,2] = PR[GP1:90,2] + 44.045;
   1:L PR[91] 10mm/sec CNT100;
   1:  PR[GP1:91,1] = PR[GP1:90,1] + -6.803;
   1:  PR[GP1:91,2] = PR[GP1:90,2] + 45.194;
   1:L PR[91] 10mm/sec CNT100;
   1:  PR[GP1:91,1] = PR[GP1:90,1] + -14.063;
   1:  PR[GP1:91,2] = PR[GP1:90,2] + 44.420;
   1:L PR[91] 10mm/sec CNT100;
   1:  PR[GP1:91,1] = PR[GP1:90,1] + -22.484;
   1:  PR[GP1:91,2] = PR[GP1:90,2] + 42.845;
   1:L PR[91] 10mm/sec CNT100;
   1:  PR[GP1:91,1] = PR[GP1:90,1] + -29.337;
   1:  PR[GP1:91,2] = PR[GP1:90,2] + 39.734;
   1:L PR[91] 10mm/sec CNT100;
   1:  PR[GP1:91,1] = PR[GP1:90,1] + -36.278;
   1:  PR[GP1:91,2] = PR[GP1:90,2] + 35.435;
   1:L PR[91] 10mm/sec CNT100;
   1:  PR[GP1:91,1] = PR[GP1:90,1] + -41.924;
   1:  PR[GP1:91,2] = PR[GP1:90,2] + 30.211;
   1:L PR[91] 10mm/sec CNT100;
   1:  PR[GP1:91,1] = PR[GP1:90,1] + -45.660;
   1:  PR[GP1:91,2] = PR[GP1:90,2] + 25.711;
   1:L PR[91] 10mm/sec CNT100;
   1:  PR[GP1:91,1] = PR[GP1:90,1] + -49.416;
   1:  PR[GP1:91,2] = PR[GP1:90,2] + 18.805;
   1:L PR[91] 10mm/sec CNT100;
   1:  PR[GP1:91,1] = PR[GP1:90,1] + -51.705;
   1:  PR[GP1:91,2] = PR[GP1:90,2] + 13.619;
   1:L PR[91] 10mm/sec CNT100;
   1:  PR[GP1:91,1] = PR[GP1:90,1] + -53.012;
   1:  PR[GP1:91,2] = PR[GP1:90,2] + 5.870;
   1:L PR[91] 10mm/sec CNT100;
   1:  PR[GP1:91,1] = PR[GP1:90,1] + -53.014;
   1:  PR[GP1:91,2] = PR[GP1:90,2] + 5.682;
   1:L PR[91] 10mm/sec CNT100;
   1:  PR[GP1:91,1] = PR[GP1:90,1] + -53.767;
   1:  PR[GP1:91,2] = PR[GP1:90,2] + 0.287;
   1:L PR[91] 10mm/sec CNT100;
   1:  PR[GP1:91,1] = PR[GP1:90,1] + -52.494;
   1:  PR[GP1:91,2] = PR[GP1:90,2] + -7.415;
   1:L PR[91] 10mm/sec CNT100;
   1:  PR[GP1:91,1] = PR[GP1:90,1] + -51.707;
   1:  PR[GP1:91,2] = PR[GP1:90,2] + -13.053;
   1:L PR[91] 10mm/sec CNT100;
   1:  PR[GP1:91,1] = PR[GP1:90,1] + -49.421;
   1:  PR[GP1:91,2] = PR[GP1:90,2] + -18.231;
   1:L PR[91] 10mm/sec CNT100;
   1:  PR[GP1:91,1] = PR[GP1:90,1] + -45.681;
   1:  PR[GP1:91,2] = PR[GP1:90,2] + -25.126;
   1:L PR[91] 10mm/sec CNT100;
   1:  PR[GP1:91,1] = PR[GP1:90,1] + -41.945;
   1:  PR[GP1:91,2] = PR[GP1:90,2] + -29.626;
   1:L PR[91] 10mm/sec CNT100;
   1:  PR[GP1:91,1] = PR[GP1:90,1] + -36.318;
   1:  PR[GP1:91,2] = PR[GP1:90,2] + -34.851;
   1:L PR[91] 10mm/sec CNT100;
   1:  PR[GP1:91,1] = PR[GP1:90,1] + -29.380;
   1:  PR[GP1:91,2] = PR[GP1:90,2] + -39.148;
   1:L PR[91] 10mm/sec CNT100;
   1:  PR[GP1:91,1] = PR[GP1:90,1] + -22.544;
   1:  PR[GP1:91,2] = PR[GP1:90,2] + -42.270;
   1:L PR[91] 10mm/sec CNT100;
   1:  PR[GP1:91,1] = PR[GP1:90,1] + -14.127;
   1:  PR[GP1:91,2] = PR[GP1:90,2] + -43.845;
   1:L PR[91] 10mm/sec CNT100;
   1:  PR[GP1:91,1] = PR[GP1:90,1] + -6.876;
   1:  PR[GP1:91,2] = PR[GP1:90,2] + -44.641;
   1:L PR[91] 10mm/sec CNT100;
   1:  PR[GP1:91,1] = PR[GP1:90,1] + -0.261;
   1:  PR[GP1:91,2] = PR[GP1:90,2] + -43.532;
   1:L PR[91] 10mm/sec CNT100;
   1:  PR[GP1:91,1] = PR[GP1:90,1] + 6.156;
   1:  PR[GP1:91,2] = PR[GP1:90,2] + -44.769;
   1:  PR[GP1:91,3] = PR[GP1:90,3] + 107.665;
   1:L PR[91] 10mm/sec CNT100;
   1:  PR[GP1:91,1] = PR[GP1:90,1] + 13.196;
   1:  PR[GP1:91,2] = PR[GP1:90,2] + -43.996;
   1:L PR[91] 10mm/sec CNT100;
   1:  PR[GP1:91,1] = PR[GP1:90,1] + 21.890;
   1:  PR[GP1:91,2] = PR[GP1:90,2] + -42.371;
   1:L PR[91] 10mm/sec CNT100;
   1:  PR[GP1:91,1] = PR[GP1:90,1] + 28.527;
   1:  PR[GP1:91,2] = PR[GP1:90,2] + -39.341;
   1:L PR[91] 10mm/sec CNT100;
   1:  PR[GP1:91,1] = PR[GP1:90,1] + 35.714;
   1:  PR[GP1:91,2] = PR[GP1:90,2] + -34.890;
   1:L PR[91] 10mm/sec CNT100;
   1:  PR[GP1:91,1] = PR[GP1:90,1] + 41.177;
   1:  PR[GP1:91,2] = PR[GP1:90,2] + -29.811;
   1:L PR[91] 10mm/sec CNT100;
   1:  PR[GP1:91,1] = PR[GP1:90,1] + 45.057;
   1:  PR[GP1:91,2] = PR[GP1:90,2] + -25.138;
   1:L PR[91] 10mm/sec CNT100;
   1:  PR[GP1:91,1] = PR[GP1:90,1] + 48.689;
   1:  PR[GP1:91,2] = PR[GP1:90,2] + -18.455;
   1:L PR[91] 10mm/sec CNT100;
   1:  PR[GP1:91,1] = PR[GP1:90,1] + 51.072;
   1:  PR[GP1:91,2] = PR[GP1:90,2] + -13.058;
   1:L PR[91] 10mm/sec CNT100;
   1:  PR[GP1:91,1] = PR[GP1:90,1] + 52.335;
   1:  PR[GP1:91,2] = PR[GP1:90,2] + -5.543;
   1:L PR[91] 10mm/sec CNT100;
   1:  PR[GP1:91,1] = PR[GP1:90,1] + 52.337;
   1:  PR[GP1:91,2] = PR[GP1:90,2] + -5.360;
   1:L PR[91] 10mm/sec CNT100;
   1:  PR[GP1:91,1] = PR[GP1:90,1] + 53.122;
   1:  PR[GP1:91,2] = PR[GP1:90,2] + 0.271;
   1:L PR[91] 10mm/sec CNT100;
   1:  PR[GP1:91,1] = PR[GP1:90,1] + 51.881;
   1:  PR[GP1:91,2] = PR[GP1:90,2] + 7.772;
   1:L PR[91] 10mm/sec CNT100;
   1:  PR[GP1:91,1] = PR[GP1:90,1] + 51.063;
   1:  PR[GP1:91,2] = PR[GP1:90,2] + 13.640;
   1:L PR[91] 10mm/sec CNT100;
   1:  PR[GP1:91,1] = PR[GP1:90,1] + 48.684;
   1:  PR[GP1:91,2] = PR[GP1:90,2] + 19.029;
   1:L PR[91] 10mm/sec CNT100;
   1:  PR[GP1:91,1] = PR[GP1:90,1] + 45.037;
   1:  PR[GP1:91,2] = PR[GP1:90,2] + 25.721;
   1:L PR[91] 10mm/sec CNT100;
   1:  PR[GP1:91,1] = PR[GP1:90,1] + 41.157;
   1:  PR[GP1:91,2] = PR[GP1:90,2] + 30.396;
   1:L PR[91] 10mm/sec CNT100;
   1:  PR[GP1:91,1] = PR[GP1:90,1] + 35.675;
   1:  PR[GP1:91,2] = PR[GP1:90,2] + 35.474;
   1:L PR[91] 10mm/sec CNT100;
   1:  PR[GP1:91,1] = PR[GP1:90,1] + 28.486;
   1:  PR[GP1:91,2] = PR[GP1:90,2] + 39.926;
   1:L PR[91] 10mm/sec CNT100;
   1:  PR[GP1:91,1] = PR[GP1:90,1] + 21.832;
   1:  PR[GP1:91,2] = PR[GP1:90,2] + 42.945;
   1:L PR[91] 10mm/sec CNT100;
   1:  PR[GP1:91,1] = PR[GP1:90,1] + 13.134;
   1:  PR[GP1:91,2] = PR[GP1:90,2] + 44.570;
   1:L PR[91] 10mm/sec CNT100;
   1:  PR[GP1:91,1] = PR[GP1:90,1] + 6.086;
   1:  PR[GP1:91,2] = PR[GP1:90,2] + 45.323;
   1:L PR[91] 10mm/sec CNT100;
   1:  PR[GP1:91,1] = PR[GP1:90,1] + -0.261;
   1:  PR[GP1:91,2] = PR[GP1:90,2] + 44.207;
   1:L PR[91] 10mm/sec CNT100;
   1:  PR[GP1:91,1] = PR[GP1:90,1] + -6.616;
   1:  PR[GP1:91,2] = PR[GP1:90,2] + 45.323;
   1:L PR[91] 10mm/sec CNT100;
   1:  PR[GP1:91,1] = PR[GP1:90,1] + -13.665;
   1:  PR[GP1:91,2] = PR[GP1:90,2] + 44.571;
   1:L PR[91] 10mm/sec CNT100;
   1:  PR[GP1:91,1] = PR[GP1:90,1] + -22.360;
   1:  PR[GP1:91,2] = PR[GP1:90,2] + 42.945;
   1:L PR[91] 10mm/sec CNT100;
   1:  PR[GP1:91,1] = PR[GP1:90,1] + -29.013;
   1:  PR[GP1:91,2] = PR[GP1:90,2] + 39.924;
   1:L PR[91] 10mm/sec CNT100;
   1:  PR[GP1:91,1] = PR[GP1:90,1] + -36.201;
   1:  PR[GP1:91,2] = PR[GP1:90,2] + 35.473;
   1:L PR[91] 10mm/sec CNT100;
   1:  PR[GP1:91,1] = PR[GP1:90,1] + -41.683;
   1:  PR[GP1:91,2] = PR[GP1:90,2] + 30.401;
   1:L PR[91] 10mm/sec CNT100;
   1:  PR[GP1:91,1] = PR[GP1:90,1] + -45.563;
   1:  PR[GP1:91,2] = PR[GP1:90,2] + 25.726;
   1:L PR[91] 10mm/sec CNT100;
   1:  PR[GP1:91,1] = PR[GP1:90,1] + -49.210;
   1:  PR[GP1:91,2] = PR[GP1:90,2] + 19.021;
   1:L PR[91] 10mm/sec CNT100;
   1:  PR[GP1:91,1] = PR[GP1:90,1] + -51.593;
   1:  PR[GP1:91,2] = PR[GP1:90,2] + 13.624;
   1:L PR[91] 10mm/sec CNT100;
   1:  PR[GP1:91,1] = PR[GP1:90,1] + -52.861;
   1:  PR[GP1:91,2] = PR[GP1:90,2] + 6.101;
   1:L PR[91] 10mm/sec CNT100;
   1:  PR[GP1:91,1] = PR[GP1:90,1] + -52.863;
   1:  PR[GP1:91,2] = PR[GP1:90,2] + 5.919;
   1:L PR[91] 10mm/sec CNT100;
   1:  PR[GP1:91,1] = PR[GP1:90,1] + -53.649;
   1:  PR[GP1:91,2] = PR[GP1:90,2] + 0.287;
   1:L PR[91] 10mm/sec CNT100;
   1:  PR[GP1:91,1] = PR[GP1:90,1] + -52.413;
   1:  PR[GP1:91,2] = PR[GP1:90,2] + -7.191;
   1:L PR[91] 10mm/sec CNT100;
   1:  PR[GP1:91,1] = PR[GP1:90,1] + -51.594;
   1:  PR[GP1:91,2] = PR[GP1:90,2] + -13.058;
   1:L PR[91] 10mm/sec CNT100;
   1:  PR[GP1:91,1] = PR[GP1:90,1] + -49.215;
   1:  PR[GP1:91,2] = PR[GP1:90,2] + -18.448;
   1:L PR[91] 10mm/sec CNT100;
   1:  PR[GP1:91,1] = PR[GP1:90,1] + -45.583;
   1:  PR[GP1:91,2] = PR[GP1:90,2] + -25.143;
   1:L PR[91] 10mm/sec CNT100;
   1:  PR[GP1:91,1] = PR[GP1:90,1] + -41.703;
   1:  PR[GP1:91,2] = PR[GP1:90,2] + -29.816;
   1:L PR[91] 10mm/sec CNT100;
   1:  PR[GP1:91,1] = PR[GP1:90,1] + -36.240;
   1:  PR[GP1:91,2] = PR[GP1:90,2] + -34.889;
   1:L PR[91] 10mm/sec CNT100;
   1:  PR[GP1:91,1] = PR[GP1:90,1] + -29.054;
   1:  PR[GP1:91,2] = PR[GP1:90,2] + -39.339;
   1:L PR[91] 10mm/sec CNT100;
   1:  PR[GP1:91,1] = PR[GP1:90,1] + -22.418;
   1:  PR[GP1:91,2] = PR[GP1:90,2] + -42.371;
   1:L PR[91] 10mm/sec CNT100;
   1:  PR[GP1:91,1] = PR[GP1:90,1] + -13.727;
   1:  PR[GP1:91,2] = PR[GP1:90,2] + -43.996;
   1:L PR[91] 10mm/sec CNT100;
   1:  PR[GP1:91,1] = PR[GP1:90,1] + -6.687;
   1:  PR[GP1:91,2] = PR[GP1:90,2] + -44.769;
   1:L PR[91] 10mm/sec CNT100;
   1:  PR[GP1:91,1] = PR[GP1:90,1] + -0.261;
   1:  PR[GP1:91,2] = PR[GP1:90,2] + -43.692;
   1:L PR[91] 10mm/sec CNT100;
   1:  PR[GP1:91,1] = PR[GP1:90,1] + 5.967;
   1:  PR[GP1:91,2] = PR[GP1:90,2] + -44.898;
   1:  PR[GP1:91,3] = PR[GP1:90,3] + 108.275;
   1:L PR[91] 10mm/sec CNT100;
   1:  PR[GP1:91,1] = PR[GP1:90,1] + 12.795;
   1:  PR[GP1:91,2] = PR[GP1:90,2] + -44.148;
   1:L PR[91] 10mm/sec CNT100;
   1:  PR[GP1:91,1] = PR[GP1:90,1] + 21.764;
   1:  PR[GP1:91,2] = PR[GP1:90,2] + -42.471;
   1:L PR[91] 10mm/sec CNT100;
   1:  PR[GP1:91,1] = PR[GP1:90,1] + 28.201;
   1:  PR[GP1:91,2] = PR[GP1:90,2] + -39.533;
   1:L PR[91] 10mm/sec CNT100;
   1:  PR[GP1:91,1] = PR[GP1:90,1] + 35.636;
   1:  PR[GP1:91,2] = PR[GP1:90,2] + -34.928;
   1:L PR[91] 10mm/sec CNT100;
   1:  PR[GP1:91,1] = PR[GP1:90,1] + 40.935;
   1:  PR[GP1:91,2] = PR[GP1:90,2] + -30.002;
   1:L PR[91] 10mm/sec CNT100;
   1:  PR[GP1:91,1] = PR[GP1:90,1] + 44.959;
   1:  PR[GP1:91,2] = PR[GP1:90,2] + -25.155;
   1:L PR[91] 10mm/sec CNT100;
   1:  PR[GP1:91,1] = PR[GP1:90,1] + 48.483;
   1:  PR[GP1:91,2] = PR[GP1:90,2] + -18.671;
   1:L PR[91] 10mm/sec CNT100;
   1:  PR[GP1:91,1] = PR[GP1:90,1] + 50.959;
   1:  PR[GP1:91,2] = PR[GP1:90,2] + -13.063;
   1:L PR[91] 10mm/sec CNT100;
   1:  PR[GP1:91,1] = PR[GP1:90,1] + 52.184;
   1:  PR[GP1:91,2] = PR[GP1:90,2] + -5.774;
   1:L PR[91] 10mm/sec CNT100;
   1:  PR[GP1:91,1] = PR[GP1:90,1] + 52.186;
   1:  PR[GP1:91,2] = PR[GP1:90,2] + -5.597;
   1:L PR[91] 10mm/sec CNT100;
   1:  PR[GP1:91,1] = PR[GP1:90,1] + 53.004;
   1:  PR[GP1:91,2] = PR[GP1:90,2] + 0.271;
   1:L PR[91] 10mm/sec CNT100;
   1:  PR[GP1:91,1] = PR[GP1:90,1] + 51.800;
   1:  PR[GP1:91,2] = PR[GP1:90,2] + 7.548;
   1:L PR[91] 10mm/sec CNT100;
   1:  PR[GP1:91,1] = PR[GP1:90,1] + 50.950;
   1:  PR[GP1:91,2] = PR[GP1:90,2] + 13.644;
   1:L PR[91] 10mm/sec CNT100;
   1:  PR[GP1:91,1] = PR[GP1:90,1] + 48.478;
   1:  PR[GP1:91,2] = PR[GP1:90,2] + 19.244;
   1:L PR[91] 10mm/sec CNT100;
   1:  PR[GP1:91,1] = PR[GP1:90,1] + 44.940;
   1:  PR[GP1:91,2] = PR[GP1:90,2] + 25.737;
   1:L PR[91] 10mm/sec CNT100;
   1:  PR[GP1:91,1] = PR[GP1:90,1] + 40.916;
   1:  PR[GP1:91,2] = PR[GP1:90,2] + 30.585;
   1:L PR[91] 10mm/sec CNT100;
   1:  PR[GP1:91,1] = PR[GP1:90,1] + 35.598;
   1:  PR[GP1:91,2] = PR[GP1:90,2] + 35.511;
   1:L PR[91] 10mm/sec CNT100;
   1:  PR[GP1:91,1] = PR[GP1:90,1] + 28.162;
   1:  PR[GP1:91,2] = PR[GP1:90,2] + 40.117;
   1:L PR[91] 10mm/sec CNT100;
   1:  PR[GP1:91,1] = PR[GP1:90,1] + 21.708;
   1:  PR[GP1:91,2] = PR[GP1:90,2] + 43.045;
   1:L PR[91] 10mm/sec CNT100;
   1:  PR[GP1:91,1] = PR[GP1:90,1] + 12.736;
   1:  PR[GP1:91,2] = PR[GP1:90,2] + 44.722;
   1:L PR[91] 10mm/sec CNT100;
   1:  PR[GP1:91,1] = PR[GP1:90,1] + 5.899;
   1:  PR[GP1:91,2] = PR[GP1:90,2] + 45.452;
   1:L PR[91] 10mm/sec CNT100;
   1:  PR[GP1:91,1] = PR[GP1:90,1] + -0.262;
   1:  PR[GP1:91,2] = PR[GP1:90,2] + 44.368;
   1:L PR[91] 10mm/sec CNT100;
   1:  PR[GP1:91,1] = PR[GP1:90,1] + -6.429;
   1:  PR[GP1:91,2] = PR[GP1:90,2] + 45.452;
   1:L PR[91] 10mm/sec CNT100;
   1:  PR[GP1:91,1] = PR[GP1:90,1] + -13.266;
   1:  PR[GP1:91,2] = PR[GP1:90,2] + 44.722;
   1:L PR[91] 10mm/sec CNT100;
   1:  PR[GP1:91,1] = PR[GP1:90,1] + -22.235;
   1:  PR[GP1:91,2] = PR[GP1:90,2] + 43.045;
   1:L PR[91] 10mm/sec CNT100;
   1:  PR[GP1:91,1] = PR[GP1:90,1] + -28.689;
   1:  PR[GP1:91,2] = PR[GP1:90,2] + 40.115;
   1:L PR[91] 10mm/sec CNT100;
   1:  PR[GP1:91,1] = PR[GP1:90,1] + -36.124;
   1:  PR[GP1:91,2] = PR[GP1:90,2] + 35.510;
   1:L PR[91] 10mm/sec CNT100;
   1:  PR[GP1:91,1] = PR[GP1:90,1] + -41.441;
   1:  PR[GP1:91,2] = PR[GP1:90,2] + 30.590;
   1:L PR[91] 10mm/sec CNT100;
   1:  PR[GP1:91,1] = PR[GP1:90,1] + -45.466;
   1:  PR[GP1:91,2] = PR[GP1:90,2] + 25.742;
   1:L PR[91] 10mm/sec CNT100;
   1:  PR[GP1:91,1] = PR[GP1:90,1] + -49.004;
   1:  PR[GP1:91,2] = PR[GP1:90,2] + 19.237;
   1:L PR[91] 10mm/sec CNT100;
   1:  PR[GP1:91,1] = PR[GP1:90,1] + -51.480;
   1:  PR[GP1:91,2] = PR[GP1:90,2] + 13.629;
   1:L PR[91] 10mm/sec CNT100;
   1:  PR[GP1:91,1] = PR[GP1:90,1] + -52.710;
   1:  PR[GP1:91,2] = PR[GP1:90,2] + 6.332;
   1:L PR[91] 10mm/sec CNT100;
   1:  PR[GP1:91,1] = PR[GP1:90,1] + -52.712;
   1:  PR[GP1:91,2] = PR[GP1:90,2] + 6.155;
   1:L PR[91] 10mm/sec CNT100;
   1:  PR[GP1:91,1] = PR[GP1:90,1] + -53.531;
   1:  PR[GP1:91,2] = PR[GP1:90,2] + 0.287;
   1:L PR[91] 10mm/sec CNT100;
   1:  PR[GP1:91,1] = PR[GP1:90,1] + -52.332;
   1:  PR[GP1:91,2] = PR[GP1:90,2] + -6.968;
   1:L PR[91] 10mm/sec CNT100;
   1:  PR[GP1:91,1] = PR[GP1:90,1] + -51.482;
   1:  PR[GP1:91,2] = PR[GP1:90,2] + -13.063;
   1:L PR[91] 10mm/sec CNT100;
   1:  PR[GP1:91,1] = PR[GP1:90,1] + -49.009;
   1:  PR[GP1:91,2] = PR[GP1:90,2] + -18.664;
   1:L PR[91] 10mm/sec CNT100;
   1:  PR[GP1:91,1] = PR[GP1:90,1] + -45.485;
   1:  PR[GP1:91,2] = PR[GP1:90,2] + -25.159;
   1:L PR[91] 10mm/sec CNT100;
   1:  PR[GP1:91,1] = PR[GP1:90,1] + -41.461;
   1:  PR[GP1:91,2] = PR[GP1:90,2] + -30.007;
   1:L PR[91] 10mm/sec CNT100;
   1:  PR[GP1:91,1] = PR[GP1:90,1] + -36.162;
   1:  PR[GP1:91,2] = PR[GP1:90,2] + -34.927;
   1:L PR[91] 10mm/sec CNT100;
   1:  PR[GP1:91,1] = PR[GP1:90,1] + -28.729;
   1:  PR[GP1:91,2] = PR[GP1:90,2] + -39.531;
   1:L PR[91] 10mm/sec CNT100;
   1:  PR[GP1:91,1] = PR[GP1:90,1] + -22.292;
   1:  PR[GP1:91,2] = PR[GP1:90,2] + -42.471;
   1:L PR[91] 10mm/sec CNT100;
   1:  PR[GP1:91,1] = PR[GP1:90,1] + -13.326;
   1:  PR[GP1:91,2] = PR[GP1:90,2] + -44.148;
   1:L PR[91] 10mm/sec CNT100;
   1:  PR[GP1:91,1] = PR[GP1:90,1] + -6.498;
   1:  PR[GP1:91,2] = PR[GP1:90,2] + -44.898;
   1:L PR[91] 10mm/sec CNT100;
   1:  PR[GP1:91,1] = PR[GP1:90,1] + -0.262;
   1:  PR[GP1:91,2] = PR[GP1:90,2] + -43.852;
   1:L PR[91] 10mm/sec CNT100;
   1:  PR[GP1:91,1] = PR[GP1:90,1] + 5.778;
   1:  PR[GP1:91,2] = PR[GP1:90,2] + -45.026;
   1:  PR[GP1:91,3] = PR[GP1:90,3] + 108.885;
   1:L PR[91] 10mm/sec CNT100;
   1:  PR[GP1:91,1] = PR[GP1:90,1] + 12.395;
   1:  PR[GP1:91,2] = PR[GP1:90,2] + -44.299;
   1:L PR[91] 10mm/sec CNT100;
   1:  PR[GP1:91,1] = PR[GP1:90,1] + 21.638;
   1:  PR[GP1:91,2] = PR[GP1:90,2] + -42.572;
   1:L PR[91] 10mm/sec CNT100;
   1:  PR[GP1:91,1] = PR[GP1:90,1] + 27.876;
   1:  PR[GP1:91,2] = PR[GP1:90,2] + -39.724;
   1:L PR[91] 10mm/sec CNT100;
   1:  PR[GP1:91,1] = PR[GP1:90,1] + 35.557;
   1:  PR[GP1:91,2] = PR[GP1:90,2] + -34.967;
   1:L PR[91] 10mm/sec CNT100;
   1:  PR[GP1:91,1] = PR[GP1:90,1] + 40.693;
   1:  PR[GP1:91,2] = PR[GP1:90,2] + -30.192;
   1:L PR[91] 10mm/sec CNT100;
   1:  PR[GP1:91,1] = PR[GP1:90,1] + 44.862;
   1:  PR[GP1:91,2] = PR[GP1:90,2] + -25.171;
   1:L PR[91] 10mm/sec CNT100;
   1:  PR[GP1:91,1] = PR[GP1:90,1] + 48.277;
   1:  PR[GP1:91,2] = PR[GP1:90,2] + -18.888;
   1:L PR[91] 10mm/sec CNT100;
   1:  PR[GP1:91,1] = PR[GP1:90,1] + 50.846;
   1:  PR[GP1:91,2] = PR[GP1:90,2] + -13.068;
   1:L PR[91] 10mm/sec CNT100;
   1:  PR[GP1:91,1] = PR[GP1:90,1] + 52.033;
   1:  PR[GP1:91,2] = PR[GP1:90,2] + -6.004;
   1:L PR[91] 10mm/sec CNT100;
   1:  PR[GP1:91,1] = PR[GP1:90,1] + 52.035;
   1:  PR[GP1:91,2] = PR[GP1:90,2] + -5.833;
   1:L PR[91] 10mm/sec CNT100;
   1:  PR[GP1:91,1] = PR[GP1:90,1] + 52.886;
   1:  PR[GP1:91,2] = PR[GP1:90,2] + 0.271;
   1:L PR[91] 10mm/sec CNT100;
   1:  PR[GP1:91,1] = PR[GP1:90,1] + 51.719;
   1:  PR[GP1:91,2] = PR[GP1:90,2] + 7.324;
   1:L PR[91] 10mm/sec CNT100;
   1:  PR[GP1:91,1] = PR[GP1:90,1] + 50.837;
   1:  PR[GP1:91,2] = PR[GP1:90,2] + 13.649;
   1:L PR[91] 10mm/sec CNT100;
   1:  PR[GP1:91,1] = PR[GP1:90,1] + 48.272;
   1:  PR[GP1:91,2] = PR[GP1:90,2] + 19.460;
   1:L PR[91] 10mm/sec CNT100;
   1:  PR[GP1:91,1] = PR[GP1:90,1] + 44.843;
   1:  PR[GP1:91,2] = PR[GP1:90,2] + 25.753;
   1:L PR[91] 10mm/sec CNT100;
   1:  PR[GP1:91,1] = PR[GP1:90,1] + 40.674;
   1:  PR[GP1:91,2] = PR[GP1:90,2] + 30.775;
   1:L PR[91] 10mm/sec CNT100;
   1:  PR[GP1:91,1] = PR[GP1:90,1] + 35.521;
   1:  PR[GP1:91,2] = PR[GP1:90,2] + 35.549;
   1:L PR[91] 10mm/sec CNT100;
   1:  PR[GP1:91,1] = PR[GP1:90,1] + 27.838;
   1:  PR[GP1:91,2] = PR[GP1:90,2] + 40.307;
   1:L PR[91] 10mm/sec CNT100;
   1:  PR[GP1:91,1] = PR[GP1:90,1] + 21.583;
   1:  PR[GP1:91,2] = PR[GP1:90,2] + 43.145;
   1:L PR[91] 10mm/sec CNT100;
   1:  PR[GP1:91,1] = PR[GP1:90,1] + 12.337;
   1:  PR[GP1:91,2] = PR[GP1:90,2] + 44.873;
   1:L PR[91] 10mm/sec CNT100;
   1:  PR[GP1:91,1] = PR[GP1:90,1] + 5.711;
   1:  PR[GP1:91,2] = PR[GP1:90,2] + 45.580;
   1:L PR[91] 10mm/sec CNT100;
   1:  PR[GP1:91,1] = PR[GP1:90,1] + -0.262;
   1:  PR[GP1:91,2] = PR[GP1:90,2] + 44.530;
   1:L PR[91] 10mm/sec CNT100;
   1:  PR[GP1:91,1] = PR[GP1:90,1] + -6.242;
   1:  PR[GP1:91,2] = PR[GP1:90,2] + 45.580;
   1:L PR[91] 10mm/sec CNT100;
   1:  PR[GP1:91,1] = PR[GP1:90,1] + -12.868;
   1:  PR[GP1:91,2] = PR[GP1:90,2] + 44.873;
   1:L PR[91] 10mm/sec CNT100;
   1:  PR[GP1:91,1] = PR[GP1:90,1] + -22.111;
   1:  PR[GP1:91,2] = PR[GP1:90,2] + 43.145;
   1:L PR[91] 10mm/sec CNT100;
   1:  PR[GP1:91,1] = PR[GP1:90,1] + -28.365;
   1:  PR[GP1:91,2] = PR[GP1:90,2] + 40.305;
   1:L PR[91] 10mm/sec CNT100;
   1:  PR[GP1:91,1] = PR[GP1:90,1] + -36.046;
   1:  PR[GP1:91,2] = PR[GP1:90,2] + 35.548;
   1:L PR[91] 10mm/sec CNT100;
   1:  PR[GP1:91,1] = PR[GP1:90,1] + -41.200;
   1:  PR[GP1:91,2] = PR[GP1:90,2] + 30.779;
   1:L PR[91] 10mm/sec CNT100;
   1:  PR[GP1:91,1] = PR[GP1:90,1] + -45.369;
   1:  PR[GP1:91,2] = PR[GP1:90,2] + 25.758;
   1:L PR[91] 10mm/sec CNT100;
   1:  PR[GP1:91,1] = PR[GP1:90,1] + -48.798;
   1:  PR[GP1:91,2] = PR[GP1:90,2] + 19.453;
   1:L PR[91] 10mm/sec CNT100;
   1:  PR[GP1:91,1] = PR[GP1:90,1] + -51.367;
   1:  PR[GP1:91,2] = PR[GP1:90,2] + 13.633;
   1:L PR[91] 10mm/sec CNT100;
   1:  PR[GP1:91,1] = PR[GP1:90,1] + -52.559;
   1:  PR[GP1:91,2] = PR[GP1:90,2] + 6.563;
   1:L PR[91] 10mm/sec CNT100;
   1:  PR[GP1:91,1] = PR[GP1:90,1] + -52.561;
   1:  PR[GP1:91,2] = PR[GP1:90,2] + 6.391;
   1:L PR[91] 10mm/sec CNT100;
   1:  PR[GP1:91,1] = PR[GP1:90,1] + -53.413;
   1:  PR[GP1:91,2] = PR[GP1:90,2] + 0.287;
   1:L PR[91] 10mm/sec CNT100;
   1:  PR[GP1:91,1] = PR[GP1:90,1] + -52.251;
   1:  PR[GP1:91,2] = PR[GP1:90,2] + -6.744;
   1:L PR[91] 10mm/sec CNT100;
   1:  PR[GP1:91,1] = PR[GP1:90,1] + -51.369;
   1:  PR[GP1:91,2] = PR[GP1:90,2] + -13.069;
   1:L PR[91] 10mm/sec CNT100;
   1:  PR[GP1:91,1] = PR[GP1:90,1] + -48.803;
   1:  PR[GP1:91,2] = PR[GP1:90,2] + -18.881;
   1:L PR[91] 10mm/sec CNT100;
   1:  PR[GP1:91,1] = PR[GP1:90,1] + -45.388;
   1:  PR[GP1:91,2] = PR[GP1:90,2] + -25.176;
   1:L PR[91] 10mm/sec CNT100;
   1:  PR[GP1:91,1] = PR[GP1:90,1] + -41.219;
   1:  PR[GP1:91,2] = PR[GP1:90,2] + -30.197;
   1:L PR[91] 10mm/sec CNT100;
   1:  PR[GP1:91,1] = PR[GP1:90,1] + -36.083;
   1:  PR[GP1:91,2] = PR[GP1:90,2] + -34.966;
   1:L PR[91] 10mm/sec CNT100;
   1:  PR[GP1:91,1] = PR[GP1:90,1] + -28.404;
   1:  PR[GP1:91,2] = PR[GP1:90,2] + -39.722;
   1:L PR[91] 10mm/sec CNT100;
   1:  PR[GP1:91,1] = PR[GP1:90,1] + -22.166;
   1:  PR[GP1:91,2] = PR[GP1:90,2] + -42.571;
   1:L PR[91] 10mm/sec CNT100;
   1:  PR[GP1:91,1] = PR[GP1:90,1] + -12.926;
   1:  PR[GP1:91,2] = PR[GP1:90,2] + -44.300;
   1:L PR[91] 10mm/sec CNT100;
   1:  PR[GP1:91,1] = PR[GP1:90,1] + -6.308;
   1:  PR[GP1:91,2] = PR[GP1:90,2] + -45.026;
   1:L PR[91] 10mm/sec CNT100;
   1:  PR[GP1:91,1] = PR[GP1:90,1] + -0.262;
   1:  PR[GP1:91,2] = PR[GP1:90,2] + -44.012;
   1:L PR[91] 10mm/sec CNT100;
   1:  PR[GP1:91,1] = PR[GP1:90,1] + 5.588;
   1:  PR[GP1:91,2] = PR[GP1:90,2] + -45.155;
   1:  PR[GP1:91,3] = PR[GP1:90,3] + 109.495;
   1:L PR[91] 10mm/sec CNT100;
   1:  PR[GP1:91,1] = PR[GP1:90,1] + 11.994;
   1:  PR[GP1:91,2] = PR[GP1:90,2] + -44.451;
   1:L PR[91] 10mm/sec CNT100;
   1:  PR[GP1:91,1] = PR[GP1:90,1] + 21.512;
   1:  PR[GP1:91,2] = PR[GP1:90,2] + -42.672;
   1:L PR[91] 10mm/sec CNT100;
   1:  PR[GP1:91,1] = PR[GP1:90,1] + 27.551;
   1:  PR[GP1:91,2] = PR[GP1:90,2] + -39.915;
   1:L PR[91] 10mm/sec CNT100;
   1:  PR[GP1:91,1] = PR[GP1:90,1] + 35.479;
   1:  PR[GP1:91,2] = PR[GP1:90,2] + -35.005;
   1:L PR[91] 10mm/sec CNT100;
   1:  PR[GP1:91,1] = PR[GP1:90,1] + 40.452;
   1:  PR[GP1:91,2] = PR[GP1:90,2] + -30.382;
   1:L PR[91] 10mm/sec CNT100;
   1:  PR[GP1:91,1] = PR[GP1:90,1] + 44.764;
   1:  PR[GP1:91,2] = PR[GP1:90,2] + -25.188;
   1:L PR[91] 10mm/sec CNT100;
   1:  PR[GP1:91,1] = PR[GP1:90,1] + 48.071;
   1:  PR[GP1:91,2] = PR[GP1:90,2] + -19.104;
   1:L PR[91] 10mm/sec CNT100;
   1:  PR[GP1:91,1] = PR[GP1:90,1] + 50.733;
   1:  PR[GP1:91,2] = PR[GP1:90,2] + -13.073;
   1:L PR[91] 10mm/sec CNT100;
   1:  PR[GP1:91,1] = PR[GP1:90,1] + 51.882;
   1:  PR[GP1:91,2] = PR[GP1:90,2] + -6.235;
   1:L PR[91] 10mm/sec CNT100;
   1:  PR[GP1:91,1] = PR[GP1:90,1] + 51.884;
   1:  PR[GP1:91,2] = PR[GP1:90,2] + -6.069;
   1:L PR[91] 10mm/sec CNT100;
   1:  PR[GP1:91,1] = PR[GP1:90,1] + 52.768;
   1:  PR[GP1:91,2] = PR[GP1:90,2] + 0.271;
   1:L PR[91] 10mm/sec CNT100;
   1:  PR[GP1:91,1] = PR[GP1:90,1] + 51.638;
   1:  PR[GP1:91,2] = PR[GP1:90,2] + 7.100;
   1:L PR[91] 10mm/sec CNT100;
   1:  PR[GP1:91,1] = PR[GP1:90,1] + 50.724;
   1:  PR[GP1:91,2] = PR[GP1:90,2] + 13.653;
   1:L PR[91] 10mm/sec CNT100;
   1:  PR[GP1:91,1] = PR[GP1:90,1] + 48.066;
   1:  PR[GP1:91,2] = PR[GP1:90,2] + 19.676;
   1:L PR[91] 10mm/sec CNT100;
   1:  PR[GP1:91,1] = PR[GP1:90,1] + 44.746;
   1:  PR[GP1:91,2] = PR[GP1:90,2] + 25.769;
   1:L PR[91] 10mm/sec CNT100;
   1:  PR[GP1:91,1] = PR[GP1:90,1] + 40.433;
   1:  PR[GP1:91,2] = PR[GP1:90,2] + 30.964;
   1:L PR[91] 10mm/sec CNT100;
   1:  PR[GP1:91,1] = PR[GP1:90,1] + 35.443;
   1:  PR[GP1:91,2] = PR[GP1:90,2] + 35.586;
   1:L PR[91] 10mm/sec CNT100;
   1:  PR[GP1:91,1] = PR[GP1:90,1] + 27.513;
   1:  PR[GP1:91,2] = PR[GP1:90,2] + 40.498;
   1:L PR[91] 10mm/sec CNT100;
   1:  PR[GP1:91,1] = PR[GP1:90,1] + 21.459;
   1:  PR[GP1:91,2] = PR[GP1:90,2] + 43.245;
   1:L PR[91] 10mm/sec CNT100;
   1:  PR[GP1:91,1] = PR[GP1:90,1] + 11.938;
   1:  PR[GP1:91,2] = PR[GP1:90,2] + 45.024;
   1:L PR[91] 10mm/sec CNT100;
   1:  PR[GP1:91,1] = PR[GP1:90,1] + 5.524;
   1:  PR[GP1:91,2] = PR[GP1:90,2] + 45.709;
   1:L PR[91] 10mm/sec CNT100;
   1:  PR[GP1:91,1] = PR[GP1:90,1] + -0.262;
   1:  PR[GP1:91,2] = PR[GP1:90,2] + 44.691;
   1:L PR[91] 10mm/sec CNT100;
   1:  PR[GP1:91,1] = PR[GP1:90,1] + -6.055;
   1:  PR[GP1:91,2] = PR[GP1:90,2] + 45.709;
   1:L PR[91] 10mm/sec CNT100;
   1:  PR[GP1:91,1] = PR[GP1:90,1] + -12.469;
   1:  PR[GP1:91,2] = PR[GP1:90,2] + 45.025;
   1:L PR[91] 10mm/sec CNT100;
   1:  PR[GP1:91,1] = PR[GP1:90,1] + -21.986;
   1:  PR[GP1:91,2] = PR[GP1:90,2] + 43.245;
   1:L PR[91] 10mm/sec CNT100;
   1:  PR[GP1:91,1] = PR[GP1:90,1] + -28.041;
   1:  PR[GP1:91,2] = PR[GP1:90,2] + 40.496;
   1:L PR[91] 10mm/sec CNT100;
   1:  PR[GP1:91,1] = PR[GP1:90,1] + -35.969;
   1:  PR[GP1:91,2] = PR[GP1:90,2] + 35.586;
   1:L PR[91] 10mm/sec CNT100;
   1:  PR[GP1:91,1] = PR[GP1:90,1] + -40.959;
   1:  PR[GP1:91,2] = PR[GP1:90,2] + 30.969;
   1:L PR[91] 10mm/sec CNT100;
   1:  PR[GP1:91,1] = PR[GP1:90,1] + -45.272;
   1:  PR[GP1:91,2] = PR[GP1:90,2] + 25.774;
   1:L PR[91] 10mm/sec CNT100;
   1:  PR[GP1:91,1] = PR[GP1:90,1] + -48.592;
   1:  PR[GP1:91,2] = PR[GP1:90,2] + 19.669;
   1:L PR[91] 10mm/sec CNT100;
   1:  PR[GP1:91,1] = PR[GP1:90,1] + -51.254;
   1:  PR[GP1:91,2] = PR[GP1:90,2] + 13.638;
   1:L PR[91] 10mm/sec CNT100;
   1:  PR[GP1:91,1] = PR[GP1:90,1] + -52.408;
   1:  PR[GP1:91,2] = PR[GP1:90,2] + 6.793;
   1:L PR[91] 10mm/sec CNT100;
   1:  PR[GP1:91,1] = PR[GP1:90,1] + -52.410;
   1:  PR[GP1:91,2] = PR[GP1:90,2] + 6.628;
   1:L PR[91] 10mm/sec CNT100;
   1:  PR[GP1:91,1] = PR[GP1:90,1] + -53.295;
   1:  PR[GP1:91,2] = PR[GP1:90,2] + 0.287;
   1:L PR[91] 10mm/sec CNT100;
   1:  PR[GP1:91,1] = PR[GP1:90,1] + -52.170;
   1:  PR[GP1:91,2] = PR[GP1:90,2] + -6.521;
   1:L PR[91] 10mm/sec CNT100;
   1:  PR[GP1:91,1] = PR[GP1:90,1] + -51.256;
   1:  PR[GP1:91,2] = PR[GP1:90,2] + -13.074;
   1:L PR[91] 10mm/sec CNT100;
   1:  PR[GP1:91,1] = PR[GP1:90,1] + -48.596;
   1:  PR[GP1:91,2] = PR[GP1:90,2] + -19.097;
   1:L PR[91] 10mm/sec CNT100;
   1:  PR[GP1:91,1] = PR[GP1:90,1] + -45.290;
   1:  PR[GP1:91,2] = PR[GP1:90,2] + -25.192;
   1:L PR[91] 10mm/sec CNT100;
   1:  PR[GP1:91,1] = PR[GP1:90,1] + -40.977;
   1:  PR[GP1:91,2] = PR[GP1:90,2] + -30.387;
   1:L PR[91] 10mm/sec CNT100;
   1:  PR[GP1:91,1] = PR[GP1:90,1] + -36.005;
   1:  PR[GP1:91,2] = PR[GP1:90,2] + -35.004;
   1:L PR[91] 10mm/sec CNT100;
   1:  PR[GP1:91,1] = PR[GP1:90,1] + -28.079;
   1:  PR[GP1:91,2] = PR[GP1:90,2] + -39.913;
   1:L PR[91] 10mm/sec CNT100;
   1:  PR[GP1:91,1] = PR[GP1:90,1] + -22.040;
   1:  PR[GP1:91,2] = PR[GP1:90,2] + -42.672;
   1:L PR[91] 10mm/sec CNT100;
   1:  PR[GP1:91,1] = PR[GP1:90,1] + -12.525;
   1:  PR[GP1:91,2] = PR[GP1:90,2] + -44.451;
   1:L PR[91] 10mm/sec CNT100;
   1:  PR[GP1:91,1] = PR[GP1:90,1] + -6.119;
   1:  PR[GP1:91,2] = PR[GP1:90,2] + -45.154;
   1:L PR[91] 10mm/sec CNT100;
   1:  PR[GP1:91,1] = PR[GP1:90,1] + -0.262;
   1:  PR[GP1:91,2] = PR[GP1:90,2] + -44.172;
   1:L PR[91] 10mm/sec CNT100;
   1:  PR[GP1:91,1] = PR[GP1:90,1] + 5.399;
   1:  PR[GP1:91,2] = PR[GP1:90,2] + -45.283;
   1:  PR[GP1:91,3] = PR[GP1:90,3] + 110.105;
   1:L PR[91] 10mm/sec CNT100;
   1:  PR[GP1:91,1] = PR[GP1:90,1] + 11.594;
   1:  PR[GP1:91,2] = PR[GP1:90,2] + -44.602;
   1:L PR[91] 10mm/sec CNT100;
   1:  PR[GP1:91,1] = PR[GP1:90,1] + 21.385;
   1:  PR[GP1:91,2] = PR[GP1:90,2] + -42.772;
   1:L PR[91] 10mm/sec CNT100;
   1:  PR[GP1:91,1] = PR[GP1:90,1] + 27.225;
   1:  PR[GP1:91,2] = PR[GP1:90,2] + -40.107;
   1:L PR[91] 10mm/sec CNT100;
   1:  PR[GP1:91,1] = PR[GP1:90,1] + 35.401;
   1:  PR[GP1:91,2] = PR[GP1:90,2] + -35.043;
   1:L PR[91] 10mm/sec CNT100;
   1:  PR[GP1:91,1] = PR[GP1:90,1] + 40.210;
   1:  PR[GP1:91,2] = PR[GP1:90,2] + -30.573;
   1:L PR[91] 10mm/sec CNT100;
   1:  PR[GP1:91,1] = PR[GP1:90,1] + 44.666;
   1:  PR[GP1:91,2] = PR[GP1:90,2] + -25.204;
   1:L PR[91] 10mm/sec CNT100;
   1:  PR[GP1:91,1] = PR[GP1:90,1] + 47.864;
   1:  PR[GP1:91,2] = PR[GP1:90,2] + -19.320;
   1:L PR[91] 10mm/sec CNT100;
   1:  PR[GP1:91,1] = PR[GP1:90,1] + 50.620;
   1:  PR[GP1:91,2] = PR[GP1:90,2] + -13.078;
   1:L PR[91] 10mm/sec CNT100;
   1:  PR[GP1:91,1] = PR[GP1:90,1] + 51.731;
   1:  PR[GP1:91,2] = PR[GP1:90,2] + -6.466;
   1:L PR[91] 10mm/sec CNT100;
   1:  PR[GP1:91,1] = PR[GP1:90,1] + 51.733;
   1:  PR[GP1:91,2] = PR[GP1:90,2] + -6.306;
   1:L PR[91] 10mm/sec CNT100;
   1:  PR[GP1:91,1] = PR[GP1:90,1] + 52.650;
   1:  PR[GP1:91,2] = PR[GP1:90,2] + 0.271;
   1:L PR[91] 10mm/sec CNT100;
   1:  PR[GP1:91,1] = PR[GP1:90,1] + 51.557;
   1:  PR[GP1:91,2] = PR[GP1:90,2] + 6.876;
   1:L PR[91] 10mm/sec CNT100;
   1:  PR[GP1:91,1] = PR[GP1:90,1] + 50.612;
   1:  PR[GP1:91,2] = PR[GP1:90,2] + 13.658;
   1:L PR[91] 10mm/sec CNT100;
   1:  PR[GP1:91,1] = PR[GP1:90,1] + 47.860;
   1:  PR[GP1:91,2] = PR[GP1:90,2] + 19.892;
   1:L PR[91] 10mm/sec CNT100;
   1:  PR[GP1:91,1] = PR[GP1:90,1] + 44.649;
   1:  PR[GP1:91,2] = PR[GP1:90,2] + 25.785;
   1:L PR[91] 10mm/sec CNT100;
   1:  PR[GP1:91,1] = PR[GP1:90,1] + 40.192;
   1:  PR[GP1:91,2] = PR[GP1:90,2] + 31.154;
   1:L PR[91] 10mm/sec CNT100;
   1:  PR[GP1:91,1] = PR[GP1:90,1] + 35.366;
   1:  PR[GP1:91,2] = PR[GP1:90,2] + 35.624;
   1:L PR[91] 10mm/sec CNT100;
   1:  PR[GP1:91,1] = PR[GP1:90,1] + 27.189;
   1:  PR[GP1:91,2] = PR[GP1:90,2] + 40.688;
   1:L PR[91] 10mm/sec CNT100;
   1:  PR[GP1:91,1] = PR[GP1:90,1] + 21.334;
   1:  PR[GP1:91,2] = PR[GP1:90,2] + 43.344;
   1:L PR[91] 10mm/sec CNT100;
   1:  PR[GP1:91,1] = PR[GP1:90,1] + 11.540;
   1:  PR[GP1:91,2] = PR[GP1:90,2] + 45.175;
   1:L PR[91] 10mm/sec CNT100;
   1:  PR[GP1:91,1] = PR[GP1:90,1] + 5.337;
   1:  PR[GP1:91,2] = PR[GP1:90,2] + 45.838;
   1:L PR[91] 10mm/sec CNT100;
   1:  PR[GP1:91,1] = PR[GP1:90,1] + -0.262;
   1:  PR[GP1:91,2] = PR[GP1:90,2] + 44.853;
   1:L PR[91] 10mm/sec CNT100;
   1:  PR[GP1:91,1] = PR[GP1:90,1] + -5.868;
   1:  PR[GP1:91,2] = PR[GP1:90,2] + 45.837;
   1:L PR[91] 10mm/sec CNT100;
   1:  PR[GP1:91,1] = PR[GP1:90,1] + -12.071;
   1:  PR[GP1:91,2] = PR[GP1:90,2] + 45.176;
   1:L PR[91] 10mm/sec CNT100;
   1:  PR[GP1:91,1] = PR[GP1:90,1] + -21.862;
   1:  PR[GP1:91,2] = PR[GP1:90,2] + 43.344;
   1:L PR[91] 10mm/sec CNT100;
   1:  PR[GP1:91,1] = PR[GP1:90,1] + -27.717;
   1:  PR[GP1:91,2] = PR[GP1:90,2] + 40.686;
   1:L PR[91] 10mm/sec CNT100;
   1:  PR[GP1:91,1] = PR[GP1:90,1] + -35.892;
   1:  PR[GP1:91,2] = PR[GP1:90,2] + 35.623;
   1:L PR[91] 10mm/sec CNT100;
   1:  PR[GP1:91,1] = PR[GP1:90,1] + -40.717;
   1:  PR[GP1:91,2] = PR[GP1:90,2] + 31.158;
   1:L PR[91] 10mm/sec CNT100;
   1:  PR[GP1:91,1] = PR[GP1:90,1] + -45.175;
   1:  PR[GP1:91,2] = PR[GP1:90,2] + 25.789;
   1:L PR[91] 10mm/sec CNT100;
   1:  PR[GP1:91,1] = PR[GP1:90,1] + -48.385;
   1:  PR[GP1:91,2] = PR[GP1:90,2] + 19.886;
   1:L PR[91] 10mm/sec CNT100;
   1:  PR[GP1:91,1] = PR[GP1:90,1] + -51.141;
   1:  PR[GP1:91,2] = PR[GP1:90,2] + 13.643;
   1:L PR[91] 10mm/sec CNT100;
   1:  PR[GP1:91,1] = PR[GP1:90,1] + -52.257;
   1:  PR[GP1:91,2] = PR[GP1:90,2] + 7.024;
   1:L PR[91] 10mm/sec CNT100;
   1:  PR[GP1:91,1] = PR[GP1:90,1] + -52.259;
   1:  PR[GP1:91,2] = PR[GP1:90,2] + 6.864;
   1:L PR[91] 10mm/sec CNT100;
   1:  PR[GP1:91,1] = PR[GP1:90,1] + -53.177;
   1:  PR[GP1:91,2] = PR[GP1:90,2] + 0.287;
   1:L PR[91] 10mm/sec CNT100;
   1:  PR[GP1:91,1] = PR[GP1:90,1] + -52.089;
   1:  PR[GP1:91,2] = PR[GP1:90,2] + -6.297;
   1:L PR[91] 10mm/sec CNT100;
   1:  PR[GP1:91,1] = PR[GP1:90,1] + -51.143;
   1:  PR[GP1:91,2] = PR[GP1:90,2] + -13.079;
   1:L PR[91] 10mm/sec CNT100;
   1:  PR[GP1:91,1] = PR[GP1:90,1] + -48.390;
   1:  PR[GP1:91,2] = PR[GP1:90,2] + -19.314;
   1:L PR[91] 10mm/sec CNT100;
   1:  PR[GP1:91,1] = PR[GP1:90,1] + -45.192;
   1:  PR[GP1:91,2] = PR[GP1:90,2] + -25.209;
   1:L PR[91] 10mm/sec CNT100;
   1:  PR[GP1:91,1] = PR[GP1:90,1] + -40.735;
   1:  PR[GP1:91,2] = PR[GP1:90,2] + -30.577;
   1:L PR[91] 10mm/sec CNT100;
   1:  PR[GP1:91,1] = PR[GP1:90,1] + -35.926;
   1:  PR[GP1:91,2] = PR[GP1:90,2] + -35.042;
   1:L PR[91] 10mm/sec CNT100;
   1:  PR[GP1:91,1] = PR[GP1:90,1] + -27.753;
   1:  PR[GP1:91,2] = PR[GP1:90,2] + -40.105;
   1:L PR[91] 10mm/sec CNT100;
   1:  PR[GP1:91,1] = PR[GP1:90,1] + -21.913;
   1:  PR[GP1:91,2] = PR[GP1:90,2] + -42.772;
   1:L PR[91] 10mm/sec CNT100;
   1:  PR[GP1:91,1] = PR[GP1:90,1] + -12.125;
   1:  PR[GP1:91,2] = PR[GP1:90,2] + -44.603;
   1:L PR[91] 10mm/sec CNT100;
   1:  PR[GP1:91,1] = PR[GP1:90,1] + -5.930;
   1:  PR[GP1:91,2] = PR[GP1:90,2] + -45.283;
   1:L PR[91] 10mm/sec CNT100;
   1:  PR[GP1:91,1] = PR[GP1:90,1] + -0.262;
   1:  PR[GP1:91,2] = PR[GP1:90,2] + -44.333;
   1:L PR[91] 10mm/sec CNT100;
   1:  PR[GP1:91,1] = PR[GP1:90,1] + 5.210;
   1:  PR[GP1:91,2] = PR[GP1:90,2] + -45.411;
   1:  PR[GP1:91,3] = PR[GP1:90,3] + 110.715;
   1:L PR[91] 10mm/sec CNT100;
   1:  PR[GP1:91,1] = PR[GP1:90,1] + 11.193;
   1:  PR[GP1:91,2] = PR[GP1:90,2] + -44.754;
   1:L PR[91] 10mm/sec CNT100;
   1:  PR[GP1:91,1] = PR[GP1:90,1] + 21.259;
   1:  PR[GP1:91,2] = PR[GP1:90,2] + -42.873;
   1:L PR[91] 10mm/sec CNT100;
   1:  PR[GP1:91,1] = PR[GP1:90,1] + 26.900;
   1:  PR[GP1:91,2] = PR[GP1:90,2] + -40.298;
   1:L PR[91] 10mm/sec CNT100;
   1:  PR[GP1:91,1] = PR[GP1:90,1] + 35.322;
   1:  PR[GP1:91,2] = PR[GP1:90,2] + -35.082;
   1:L PR[91] 10mm/sec CNT100;
   1:  PR[GP1:91,1] = PR[GP1:90,1] + 39.968;
   1:  PR[GP1:91,2] = PR[GP1:90,2] + -30.763;
   1:L PR[91] 10mm/sec CNT100;
   1:  PR[GP1:91,1] = PR[GP1:90,1] + 44.569;
   1:  PR[GP1:91,2] = PR[GP1:90,2] + -25.221;
   1:L PR[91] 10mm/sec CNT100;
   1:  PR[GP1:91,1] = PR[GP1:90,1] + 47.658;
   1:  PR[GP1:91,2] = PR[GP1:90,2] + -19.536;
   1:L PR[91] 10mm/sec CNT100;
   1:  PR[GP1:91,1] = PR[GP1:90,1] + 50.507;
   1:  PR[GP1:91,2] = PR[GP1:90,2] + -13.083;
   1:L PR[91] 10mm/sec CNT100;
   1:  PR[GP1:91,1] = PR[GP1:90,1] + 51.580;
   1:  PR[GP1:91,2] = PR[GP1:90,2] + -6.697;
   1:L PR[91] 10mm/sec CNT100;
   1:  PR[GP1:91,1] = PR[GP1:90,1] + 51.582;
   1:  PR[GP1:91,2] = PR[GP1:90,2] + -6.542;
   1:L PR[91] 10mm/sec CNT100;
   1:  PR[GP1:91,1] = PR[GP1:90,1] + 52.532;
   1:  PR[GP1:91,2] = PR[GP1:90,2] + 0.271;
   1:L PR[91] 10mm/sec CNT100;
   1:  PR[GP1:91,1] = PR[GP1:90,1] + 51.477;
   1:  PR[GP1:91,2] = PR[GP1:90,2] + 6.652;
   1:L PR[91] 10mm/sec CNT100;
   1:  PR[GP1:91,1] = PR[GP1:90,1] + 50.499;
   1:  PR[GP1:91,2] = PR[GP1:90,2] + 13.662;
   1:L PR[91] 10mm/sec CNT100;
   1:  PR[GP1:91,1] = PR[GP1:90,1] + 47.653;
   1:  PR[GP1:91,2] = PR[GP1:90,2] + 20.108;
   1:L PR[91] 10mm/sec CNT100;
   1:  PR[GP1:91,1] = PR[GP1:90,1] + 44.552;
   1:  PR[GP1:91,2] = PR[GP1:90,2] + 25.801;
   1:L PR[91] 10mm/sec CNT100;
   1:  PR[GP1:91,1] = PR[GP1:90,1] + 39.951;
   1:  PR[GP1:91,2] = PR[GP1:90,2] + 31.343;
   1:L PR[91] 10mm/sec CNT100;
   1:  PR[GP1:91,1] = PR[GP1:90,1] + 35.289;
   1:  PR[GP1:91,2] = PR[GP1:90,2] + 35.661;
   1:L PR[91] 10mm/sec CNT100;
   1:  PR[GP1:91,1] = PR[GP1:90,1] + 26.865;
   1:  PR[GP1:91,2] = PR[GP1:90,2] + 40.879;
   1:L PR[91] 10mm/sec CNT100;
   1:  PR[GP1:91,1] = PR[GP1:90,1] + 21.209;
   1:  PR[GP1:91,2] = PR[GP1:90,2] + 43.444;
   1:L PR[91] 10mm/sec CNT100;
   1:  PR[GP1:91,1] = PR[GP1:90,1] + 11.141;
   1:  PR[GP1:91,2] = PR[GP1:90,2] + 45.326;
   1:L PR[91] 10mm/sec CNT100;
   1:  PR[GP1:91,1] = PR[GP1:90,1] + 5.150;
   1:  PR[GP1:91,2] = PR[GP1:90,2] + 45.966;
   1:L PR[91] 10mm/sec CNT100;
   1:  PR[GP1:91,1] = PR[GP1:90,1] + -0.262;
   1:  PR[GP1:91,2] = PR[GP1:90,2] + 45.014;
   1:L PR[91] 10mm/sec CNT100;
   1:  PR[GP1:91,1] = PR[GP1:90,1] + -5.681;
   1:  PR[GP1:91,2] = PR[GP1:90,2] + 45.966;
   1:L PR[91] 10mm/sec CNT100;
   1:  PR[GP1:91,1] = PR[GP1:90,1] + -11.672;
   1:  PR[GP1:91,2] = PR[GP1:90,2] + 45.327;
   1:L PR[91] 10mm/sec CNT100;
   1:  PR[GP1:91,1] = PR[GP1:90,1] + -21.737;
   1:  PR[GP1:91,2] = PR[GP1:90,2] + 43.444;
   1:L PR[91] 10mm/sec CNT100;
   1:  PR[GP1:91,1] = PR[GP1:90,1] + -27.393;
   1:  PR[GP1:91,2] = PR[GP1:90,2] + 40.877;
   1:L PR[91] 10mm/sec CNT100;
   1:  PR[GP1:91,1] = PR[GP1:90,1] + -35.815;
   1:  PR[GP1:91,2] = PR[GP1:90,2] + 35.661;
   1:L PR[91] 10mm/sec CNT100;
   1:  PR[GP1:91,1] = PR[GP1:90,1] + -40.476;
   1:  PR[GP1:91,2] = PR[GP1:90,2] + 31.348;
   1:L PR[91] 10mm/sec CNT100;
   1:  PR[GP1:91,1] = PR[GP1:90,1] + -45.078;
   1:  PR[GP1:91,2] = PR[GP1:90,2] + 25.805;
   1:L PR[91] 10mm/sec CNT100;
   1:  PR[GP1:91,1] = PR[GP1:90,1] + -48.179;
   1:  PR[GP1:91,2] = PR[GP1:90,2] + 20.102;
   1:L PR[91] 10mm/sec CNT100;
   1:  PR[GP1:91,1] = PR[GP1:90,1] + -51.029;
   1:  PR[GP1:91,2] = PR[GP1:90,2] + 13.648;
   1:L PR[91] 10mm/sec CNT100;
   1:  PR[GP1:91,1] = PR[GP1:90,1] + -52.107;
   1:  PR[GP1:91,2] = PR[GP1:90,2] + 7.255;
   1:L PR[91] 10mm/sec CNT100;
   1:  PR[GP1:91,1] = PR[GP1:90,1] + -52.108;
   1:  PR[GP1:91,2] = PR[GP1:90,2] + 7.100;
   1:L PR[91] 10mm/sec CNT100;
   1:  PR[GP1:91,1] = PR[GP1:90,1] + -53.059;
   1:  PR[GP1:91,2] = PR[GP1:90,2] + 0.287;
   1:L PR[91] 10mm/sec CNT100;
   1:  PR[GP1:91,1] = PR[GP1:90,1] + -52.008;
   1:  PR[GP1:91,2] = PR[GP1:90,2] + -6.074;
   1:L PR[91] 10mm/sec CNT100;
   1:  PR[GP1:91,1] = PR[GP1:90,1] + -51.030;
   1:  PR[GP1:91,2] = PR[GP1:90,2] + -13.085;
   1:L PR[91] 10mm/sec CNT100;
   1:  PR[GP1:91,1] = PR[GP1:90,1] + -48.184;
   1:  PR[GP1:91,2] = PR[GP1:90,2] + -19.530;
   1:L PR[91] 10mm/sec CNT100;
   1:  PR[GP1:91,1] = PR[GP1:90,1] + -45.094;
   1:  PR[GP1:91,2] = PR[GP1:90,2] + -25.225;
   1:L PR[91] 10mm/sec CNT100;
   1:  PR[GP1:91,1] = PR[GP1:90,1] + -40.493;
   1:  PR[GP1:91,2] = PR[GP1:90,2] + -30.768;
   1:L PR[91] 10mm/sec CNT100;
   1:  PR[GP1:91,1] = PR[GP1:90,1] + -35.848;
   1:  PR[GP1:91,2] = PR[GP1:90,2] + -35.081;
   1:L PR[91] 10mm/sec CNT100;
   1:  PR[GP1:91,1] = PR[GP1:90,1] + -27.428;
   1:  PR[GP1:91,2] = PR[GP1:90,2] + -40.296;
   1:L PR[91] 10mm/sec CNT100;
   1:  PR[GP1:91,1] = PR[GP1:90,1] + -21.787;
   1:  PR[GP1:91,2] = PR[GP1:90,2] + -42.873;
   1:L PR[91] 10mm/sec CNT100;
   1:  PR[GP1:91,1] = PR[GP1:90,1] + -11.725;
   1:  PR[GP1:91,2] = PR[GP1:90,2] + -44.755;
   1:L PR[91] 10mm/sec CNT100;
   1:  PR[GP1:91,1] = PR[GP1:90,1] + -5.741;
   1:  PR[GP1:91,2] = PR[GP1:90,2] + -45.411;
   1:L PR[91] 10mm/sec CNT100;
   1:  PR[GP1:91,1] = PR[GP1:90,1] + -0.262;
   1:  PR[GP1:91,2] = PR[GP1:90,2] + -44.493;
   1:L PR[91] 10mm/sec CNT100;
   1:  PR[GP1:91,1] = PR[GP1:90,1] + 5.020;
   1:  PR[GP1:91,2] = PR[GP1:90,2] + -45.540;
   1:  PR[GP1:91,3] = PR[GP1:90,3] + 111.325;
   1:L PR[91] 10mm/sec CNT100;
   1:  PR[GP1:91,1] = PR[GP1:90,1] + 10.793;
   1:  PR[GP1:91,2] = PR[GP1:90,2] + -44.906;
   1:L PR[91] 10mm/sec CNT100;
   1:  PR[GP1:91,1] = PR[GP1:90,1] + 21.133;
   1:  PR[GP1:91,2] = PR[GP1:90,2] + -42.973;
   1:L PR[91] 10mm/sec CNT100;
   1:  PR[GP1:91,1] = PR[GP1:90,1] + 26.574;
   1:  PR[GP1:91,2] = PR[GP1:90,2] + -40.489;
   1:L PR[91] 10mm/sec CNT100;
   1:  PR[GP1:91,1] = PR[GP1:90,1] + 35.244;
   1:  PR[GP1:91,2] = PR[GP1:90,2] + -35.120;
   1:L PR[91] 10mm/sec CNT100;
   1:  PR[GP1:91,1] = PR[GP1:90,1] + 39.726;
   1:  PR[GP1:91,2] = PR[GP1:90,2] + -30.954;
   1:L PR[91] 10mm/sec CNT100;
   1:  PR[GP1:91,1] = PR[GP1:90,1] + 44.471;
   1:  PR[GP1:91,2] = PR[GP1:90,2] + -25.238;
   1:L PR[91] 10mm/sec CNT100;
   1:  PR[GP1:91,1] = PR[GP1:90,1] + 47.452;
   1:  PR[GP1:91,2] = PR[GP1:90,2] + -19.753;
   1:L PR[91] 10mm/sec CNT100;
   1:  PR[GP1:91,1] = PR[GP1:90,1] + 50.394;
   1:  PR[GP1:91,2] = PR[GP1:90,2] + -13.088;
   1:L PR[91] 10mm/sec CNT100;
   1:  PR[GP1:91,1] = PR[GP1:90,1] + 51.429;
   1:  PR[GP1:91,2] = PR[GP1:90,2] + -6.927;
   1:L PR[91] 10mm/sec CNT100;
   1:  PR[GP1:91,1] = PR[GP1:90,1] + 51.431;
   1:  PR[GP1:91,2] = PR[GP1:90,2] + -6.778;
   1:L PR[91] 10mm/sec CNT100;
   1:  PR[GP1:91,1] = PR[GP1:90,1] + 52.414;
   1:  PR[GP1:91,2] = PR[GP1:90,2] + 0.271;
   1:L PR[91] 10mm/sec CNT100;
   1:  PR[GP1:91,1] = PR[GP1:90,1] + 51.396;
   1:  PR[GP1:91,2] = PR[GP1:90,2] + 6.428;
   1:L PR[91] 10mm/sec CNT100;
   1:  PR[GP1:91,1] = PR[GP1:90,1] + 50.386;
   1:  PR[GP1:91,2] = PR[GP1:90,2] + 13.667;
   1:L PR[91] 10mm/sec CNT100;
   1:  PR[GP1:91,1] = PR[GP1:90,1] + 47.447;
   1:  PR[GP1:91,2] = PR[GP1:90,2] + 20.323;
   1:L PR[91] 10mm/sec CNT100;
   1:  PR[GP1:91,1] = PR[GP1:90,1] + 44.455;
   1:  PR[GP1:91,2] = PR[GP1:90,2] + 25.817;
   1:L PR[91] 10mm/sec CNT100;
   1:  PR[GP1:91,1] = PR[GP1:90,1] + 39.709;
   1:  PR[GP1:91,2] = PR[GP1:90,2] + 31.533;
   1:L PR[91] 10mm/sec CNT100;
   1:  PR[GP1:91,1] = PR[GP1:90,1] + 35.212;
   1:  PR[GP1:91,2] = PR[GP1:90,2] + 35.699;
   1:L PR[91] 10mm/sec CNT100;
   1:  PR[GP1:91,1] = PR[GP1:90,1] + 26.541;
   1:  PR[GP1:91,2] = PR[GP1:90,2] + 41.069;
   1:L PR[91] 10mm/sec CNT100;
   1:  PR[GP1:91,1] = PR[GP1:90,1] + 21.085;
   1:  PR[GP1:91,2] = PR[GP1:90,2] + 43.544;
   1:L PR[91] 10mm/sec CNT100;
   1:  PR[GP1:91,1] = PR[GP1:90,1] + 10.742;
   1:  PR[GP1:91,2] = PR[GP1:90,2] + 45.477;
   1:L PR[91] 10mm/sec CNT100;
   1:  PR[GP1:91,1] = PR[GP1:90,1] + 4.963;
   1:  PR[GP1:91,2] = PR[GP1:90,2] + 46.095;
   1:L PR[91] 10mm/sec CNT100;
   1:  PR[GP1:91,1] = PR[GP1:90,1] + -0.262;
   1:  PR[GP1:91,2] = PR[GP1:90,2] + 45.176;
   1:L PR[91] 10mm/sec CNT100;
   1:  PR[GP1:91,1] = PR[GP1:90,1] + -5.494;
   1:  PR[GP1:91,2] = PR[GP1:90,2] + 46.094;
   1:L PR[91] 10mm/sec CNT100;
   1:  PR[GP1:91,1] = PR[GP1:90,1] + -11.274;
   1:  PR[GP1:91,2] = PR[GP1:90,2] + 45.478;
   1:L PR[91] 10mm/sec CNT100;
   1:  PR[GP1:91,1] = PR[GP1:90,1] + -21.613;
   1:  PR[GP1:91,2] = PR[GP1:90,2] + 43.544;
   1:L PR[91] 10mm/sec CNT100;
   1:  PR[GP1:91,1] = PR[GP1:90,1] + -27.069;
   1:  PR[GP1:91,2] = PR[GP1:90,2] + 41.067;
   1:L PR[91] 10mm/sec CNT100;
   1:  PR[GP1:91,1] = PR[GP1:90,1] + -35.738;
   1:  PR[GP1:91,2] = PR[GP1:90,2] + 35.698;
   1:L PR[91] 10mm/sec CNT100;
   1:  PR[GP1:91,1] = PR[GP1:90,1] + -40.235;
   1:  PR[GP1:91,2] = PR[GP1:90,2] + 31.537;
   1:L PR[91] 10mm/sec CNT100;
   1:  PR[GP1:91,1] = PR[GP1:90,1] + -44.980;
   1:  PR[GP1:91,2] = PR[GP1:90,2] + 25.821;
   1:L PR[91] 10mm/sec CNT100;
   1:  PR[GP1:91,1] = PR[GP1:90,1] + -47.973;
   1:  PR[GP1:91,2] = PR[GP1:90,2] + 20.318;
   1:L PR[91] 10mm/sec CNT100;
   1:  PR[GP1:91,1] = PR[GP1:90,1] + -50.916;
   1:  PR[GP1:91,2] = PR[GP1:90,2] + 13.653;
   1:L PR[91] 10mm/sec CNT100;
   1:  PR[GP1:91,1] = PR[GP1:90,1] + -51.956;
   1:  PR[GP1:91,2] = PR[GP1:90,2] + 7.485;
   1:L PR[91] 10mm/sec CNT100;
   1:  PR[GP1:91,1] = PR[GP1:90,1] + -51.957;
   1:  PR[GP1:91,2] = PR[GP1:90,2] + 7.337;
   1:L PR[91] 10mm/sec CNT100;
   1:  PR[GP1:91,1] = PR[GP1:90,1] + -52.941;
   1:  PR[GP1:91,2] = PR[GP1:90,2] + 0.287;
   1:L PR[91] 10mm/sec CNT100;
   1:  PR[GP1:91,1] = PR[GP1:90,1] + -51.926;
   1:  PR[GP1:91,2] = PR[GP1:90,2] + -5.850;
   1:L PR[91] 10mm/sec CNT100;
   1:  PR[GP1:91,1] = PR[GP1:90,1] + -50.917;
   1:  PR[GP1:91,2] = PR[GP1:90,2] + -13.090;
   1:L PR[91] 10mm/sec CNT100;
   1:  PR[GP1:91,1] = PR[GP1:90,1] + -47.978;
   1:  PR[GP1:91,2] = PR[GP1:90,2] + -19.747;
   1:L PR[91] 10mm/sec CNT100;
   1:  PR[GP1:91,1] = PR[GP1:90,1] + -44.997;
   1:  PR[GP1:91,2] = PR[GP1:90,2] + -25.242;
   1:L PR[91] 10mm/sec CNT100;
   1:  PR[GP1:91,1] = PR[GP1:90,1] + -40.251;
   1:  PR[GP1:91,2] = PR[GP1:90,2] + -30.958;
   1:L PR[91] 10mm/sec CNT100;
   1:  PR[GP1:91,1] = PR[GP1:90,1] + -35.770;
   1:  PR[GP1:91,2] = PR[GP1:90,2] + -35.119;
   1:L PR[91] 10mm/sec CNT100;
   1:  PR[GP1:91,1] = PR[GP1:90,1] + -27.103;
   1:  PR[GP1:91,2] = PR[GP1:90,2] + -40.487;
   1:L PR[91] 10mm/sec CNT100;
   1:  PR[GP1:91,1] = PR[GP1:90,1] + -21.661;
   1:  PR[GP1:91,2] = PR[GP1:90,2] + -42.973;
   1:L PR[91] 10mm/sec CNT100;
   1:  PR[GP1:91,1] = PR[GP1:90,1] + -11.324;
   1:  PR[GP1:91,2] = PR[GP1:90,2] + -44.906;
   1:L PR[91] 10mm/sec CNT100;
   1:  PR[GP1:91,1] = PR[GP1:90,1] + -5.552;
   1:  PR[GP1:91,2] = PR[GP1:90,2] + -45.540;
   1:L PR[91] 10mm/sec CNT100;
   1:  PR[GP1:91,1] = PR[GP1:90,1] + -0.262;
   1:  PR[GP1:91,2] = PR[GP1:90,2] + -44.653;
   1:L PR[91] 10mm/sec CNT100;
   1:  PR[GP1:91,1] = PR[GP1:90,1] + 4.831;
   1:  PR[GP1:91,2] = PR[GP1:90,2] + -45.668;
   1:  PR[GP1:91,3] = PR[GP1:90,3] + 111.935;
   1:L PR[91] 10mm/sec CNT100;
   1:  PR[GP1:91,1] = PR[GP1:90,1] + 10.392;
   1:  PR[GP1:91,2] = PR[GP1:90,2] + -45.057;
   1:L PR[91] 10mm/sec CNT100;
   1:  PR[GP1:91,1] = PR[GP1:90,1] + 21.007;
   1:  PR[GP1:91,2] = PR[GP1:90,2] + -43.073;
   1:L PR[91] 10mm/sec CNT100;
   1:  PR[GP1:91,1] = PR[GP1:90,1] + 26.249;
   1:  PR[GP1:91,2] = PR[GP1:90,2] + -40.680;
   1:L PR[91] 10mm/sec CNT100;
   1:  PR[GP1:91,1] = PR[GP1:90,1] + 35.166;
   1:  PR[GP1:91,2] = PR[GP1:90,2] + -35.158;
   1:L PR[91] 10mm/sec CNT100;
   1:  PR[GP1:91,1] = PR[GP1:90,1] + 39.484;
   1:  PR[GP1:91,2] = PR[GP1:90,2] + -31.144;
   1:L PR[91] 10mm/sec CNT100;
   1:  PR[GP1:91,1] = PR[GP1:90,1] + 44.373;
   1:  PR[GP1:91,2] = PR[GP1:90,2] + -25.254;
   1:L PR[91] 10mm/sec CNT100;
   1:  PR[GP1:91,1] = PR[GP1:90,1] + 47.246;
   1:  PR[GP1:91,2] = PR[GP1:90,2] + -19.969;
   1:L PR[91] 10mm/sec CNT100;
   1:  PR[GP1:91,1] = PR[GP1:90,1] + 50.281;
   1:  PR[GP1:91,2] = PR[GP1:90,2] + -13.093;
   1:L PR[91] 10mm/sec CNT100;
   1:  PR[GP1:91,1] = PR[GP1:90,1] + 51.278;
   1:  PR[GP1:91,2] = PR[GP1:90,2] + -7.158;
   1:L PR[91] 10mm/sec CNT100;
